(* CODESYS project SUZUKI.project
   Title: ifmCR711S_TemplateProject
   Company: ifm electronic
   Version: 2.4.13.0
   Description: Project template with CR711S configured 2.25MByte Standard 2.25MByte Safety

Project tree, tasks and I/O mapping:
  StandardPLC : CR711S Standard, ifm electronic, order no. CR711S, version 3.0.0.1
    application Application
      libraries: Standard, * (System); Util, * (System); SysMem, * (System); ifmR360-3, 1.1.1.0 (ifm electronic); SysTimeCore, 3.5.5.0 (System); SysFile, 3.5.9.0 (System); SysCom, 3.5.5.0 (System); ifmOutHBridge, 2.3.0.0 (ifm electronic); CAA CiA 405, 3.5.8.0 (CAA Technical Workgroup); TCP, 3.5.9.50 (3S - Smart Software Solutions GmbH)
      task Tarea_Can (cyclic, interval t#10ms, priority 0) calls nothing
      task Tarea_Codigo (cyclic, interval t#20ms, priority 1, watchdog t#200ms x 1) calls PLC_PRG
      CÓDIGO/
        program SALIDAS [ST]
        Seguridades/
          program Laser_Seguridad [ST]
          program Setas_Seguridad [ST]
          program Campos_Laser [ST]
        program SUPERVISOR [ST]
        Data types/
          data type AccionLevas
          data type ENTRADAS_PLC
          data type EstadoSecuenciaCarga
          data type CamposLaser
          data type ControlVelocidad
          data type ENTRADAS_AGV
          data type SALIDAS_PLC
          data type OperativaARealizar
          data type EstadoEframe
          data type VelocidadPorTramo
        AUX_IFM/
          function block fb_InputAddConf_sp_ST_V02 [FBD]
          function block fb_OutputGroupAddConf_sp_ST_V02 [FBD]
          function block fb_OutputAnaAddConf_sp_ST_V02 [FBD]
          function block fb_OutputAddConf_sp_ST_V02 [FBD]
        program ESTADOS [ST]
        Sub ACCIONES/
          program ACC03_ControlLevas [ST]
          program ACC00_SalidasDesactivadas [ST]
          program ACC02_ControlAutomatico [ST]
          program ACC01_ControlManual [ST]
        program IMAGENES [ST]
        program PLC_PRG [ST]
        program PARAMETRIZACION [ST]
        Sub Comunicacion/
          program C41 [ST]
          function block COM00_DispositivoCAN_FB [ST]
          program C40 [ST]
        Sub Temporizacion/
          program TEMP00_TiempoInicio [ST]
        program ACCIONES [ST]
        program COMUNICACION_CAN [ST]
        IO/
          program OUT01_WIRED_OUTPUTS [ST]
          program IN01_WIRED_INPUTS [ST]
        Sub Dispositivos/
          function block DISP01_CntrlExtensionGeneral_FB [ST]
          program DISP02_Indicadores [ST]
          program DISP03_EncoderTeaching [ST]
      Global Variables/
        global variables Variables_globales_persistentes
        data type MatrizPDO
        data type MatrizPDOUSINT
        data type SpCanOpenNode
        global variables Global_Variables
      Visualizaciones/
        trace Anomalia (task Tarea_Codigo): COMUNICACION_CAN.O_EstadoCAN.0
    Communication : Communication, ifm electronic, version 3.0.0.1
      Ethernet : Ethernet, ifm electronic, version 3.0.0.1
      CAN : CAN, ifm electronic, version 3.0.0.1
        ifmCANbus : ifmCANbus, ifm electronic, version 1.0.0.0
            settings: NetID = 2
          CANopen_Manager : CANopen_Manager, 3S - Smart Software Solutions GmbH, version 3.5.16.0
              settings: Sync CycleTime in Microseconds = 10000; Enable Sync generation = TRUE; Synchronous Window Length = 201010; NMT Start All = TRUE; Heartbeat in Milliseconds = 100; Heartbeat Node ID = 1; CANopen NodeID = 1; ConfigVersion = 50659584
            UCD_Encoder_Series : UCD Encoder Series, Posital GmbH, order no. UCD-CA01B-xxxx-xxxx-xxx, version Revision=16#00010000, FileVersion=1.1, File=UCD-CAx1B-xxxx-xxxx-xxx_V1R4.eds
                settings: General Options.Optional Device = TRUE; General Options.Reset Node = FALSE; NODEIDSAVED = 32; SDO Timeout = 1000000; PDO_Autoconfig = FALSE; EXPERTSETTINGS = True; Sync-General Parameters.Sync-COBID = 16#00000080; Sync-General Parameters.Communication Cycle Period = 16#00002710 usec; Synchronous Window Length = 16#00031132; SubIndex for reset node = 1; Emergency-General Parameters.Emergency enabled = FALSE; Emergency-General Parameters.Emergency COBID = 16#000000A0; Heartbeat-Producer Time = 100; PDO 16#1800.COBID = 16#000001A0; Process by CANopenManager = TRUE; PDO 16#1801.COBID = 16#000002A0; PDO 16#1801.Transmission Type = 16#01; Process by CANopenManager = TRUE; Heartbeat-Consuming1.Heartbeat-Time = 150 ms; Position value.Subindex = 16#00; Position value.Subindex = 16#00; SDO List.Set COB-ID sync.Index = 16#1005; SDO List.Set COB-ID sync.Subindex = 16#00; SDO List.Set COB-ID sync.Value = 16#00000080; SDO List.Set COB-ID sync.Size = 32; SDO List.Set COB-ID sync.AbortIfError = FALSE; SDO List.Set COB-ID sync.JumpToLine = FALSE; SDO List.Set COB-ID sync.Line = 0; SDO List.Set communication cycle period.Index = 16#1006; SDO List.Set communication cycle period.Subindex = 16#00; SDO List.Set communication cycle period.Value = 16#00002710; SDO List.Set communication cycle period.Size = 32; SDO List.Set communication cycle period.AbortIfError = FALSE; SDO List.Set communication cycle period.JumpToLine = FALSE; SDO List.Set communication cycle period.Line = 0; SDO List.Set synchronous window length.Index = 16#1007; SDO List.Set synchronous window length.Subindex = 16#00; SDO List.Set synchronous window length.Value = 16#00031132; SDO List.Set synchronous window length.Size = 32; SDO List.Set synchronous window length.AbortIfError = FALSE;
                  SDO List.Set synchronous window length.JumpToLine = FALSE; SDO List.Set synchronous window length.Line = 0; SDO List.Disable TIME.Index = 16#1012; SDO List.Disable TIME.Subindex = 16#00; SDO List.Disable TIME.Value = 16#00000100; SDO List.Disable TIME.Size = 32; SDO List.Disable TIME.AbortIfError = FALSE; SDO List.Disable TIME.JumpToLine = FALSE; SDO List.Disable TIME.Line = 0; SDO List.Set Guardtime.Index = 16#100C; SDO List.Set Guardtime.Subindex = 16#00; SDO List.Set Guardtime.Value = 16#00000000; SDO List.Set Guardtime.Size = 16; SDO List.Set Guardtime.AbortIfError = FALSE; SDO List.Set Guardtime.JumpToLine = FALSE; SDO List.Set Guardtime.Line = 0; SDO List.Set Lifetime.Index = 16#100D; SDO List.Set Lifetime.Subindex = 16#00; SDO List.Set Lifetime.Value = 16#00000000; SDO List.Set Lifetime.Size = 8; SDO List.Set Lifetime.AbortIfError = FALSE; SDO List.Set Lifetime.JumpToLine = FALSE; SDO List.Set Lifetime.Line = 0; SDO List.Set Heartbeat Consumer.Index = 16#1016; SDO List.Set Heartbeat Consumer.Subindex = 16#01; SDO List.Set Heartbeat Consumer.Value = 16#00010096; SDO List.Set Heartbeat Consumer.Size = 32; SDO List.Set Heartbeat Consumer.AbortIfError = FALSE; SDO List.Set Heartbeat Consumer.JumpToLine = FALSE; SDO List.Set Heartbeat Consumer.Line = 0; SDO List.Set Heartbeat Producer.Index = 16#1017; SDO List.Set Heartbeat Producer.Subindex = 16#00; SDO List.Set Heartbeat Producer.Value = 16#00000064; SDO List.Set Heartbeat Producer.Size = 16; SDO List.Set Heartbeat Producer.AbortIfError = FALSE; SDO List.Set Heartbeat Producer.JumpToLine = FALSE; SDO List.Set Heartbeat Producer.Line = 0; SDO List.Disable PDO.Index = 16#1800; SDO List.Disable PDO.Subindex = 16#01; SDO List.Disable PDO.Value = 16#800001A0;
                  SDO List.Disable PDO.Size = 32; SDO List.Disable PDO.AbortIfError = FALSE; SDO List.Disable PDO.JumpToLine = FALSE; SDO List.Disable PDO.Line = 0; SDO List.Set transmission type.Index = 16#1800; SDO List.Set transmission type.Subindex = 16#02; SDO List.Set transmission type.Value = 16#FE; SDO List.Set transmission type.Size = 8; SDO List.Set transmission type.AbortIfError = FALSE; SDO List.Set transmission type.JumpToLine = FALSE; SDO List.Set transmission type.Line = 0; SDO List.Set inhibit time.Index = 16#1800; SDO List.Set inhibit time.Subindex = 16#03; SDO List.Set inhibit time.Value = 16#0000; SDO List.Set inhibit time.Size = 16; SDO List.Set inhibit time.AbortIfError = FALSE; SDO List.Set inhibit time.JumpToLine = FALSE; SDO List.Set inhibit time.Line = 0; SDO List.Set event time.Index = 16#1800; SDO List.Set event time.Subindex = 16#05; SDO List.Set event time.Value = 16#0000; SDO List.Set event time.Size = 16; SDO List.Set event time.AbortIfError = FALSE; SDO List.Set event time.JumpToLine = FALSE; SDO List.Set event time.Line = 0; SDO List.Clear pdo mapping.Index = 16#1A00; SDO List.Clear pdo mapping.Subindex = 16#00; SDO List.Clear pdo mapping.Value = 16#0; SDO List.Clear pdo mapping.Size = 8; SDO List.Clear pdo mapping.AbortIfError = FALSE; SDO List.Clear pdo mapping.JumpToLine = FALSE; SDO List.Clear pdo mapping.Line = 0; SDO List.Set Mapping.Index = 16#1A00; SDO List.Set Mapping.Subindex = 16#01; SDO List.Set Mapping.Value = 16#60040020; SDO List.Set Mapping.Size = 32; SDO List.Set Mapping.AbortIfError = FALSE; SDO List.Set Mapping.JumpToLine = FALSE; SDO List.Set Mapping.Line = 0; SDO List.Set number of mappings.Index = 16#1A00;
                  SDO List.Set number of mappings.Subindex = 16#00; SDO List.Set number of mappings.Value = 16#01; SDO List.Set number of mappings.Size = 8; SDO List.Set number of mappings.AbortIfError = FALSE; SDO List.Set number of mappings.JumpToLine = FALSE; SDO List.Set number of mappings.Line = 0; SDO List.Set and enable COB-ID.Index = 16#1800; SDO List.Set and enable COB-ID.Subindex = 16#01; SDO List.Set and enable COB-ID.Value = 16#000001A0; SDO List.Set and enable COB-ID.Size = 32; SDO List.Set and enable COB-ID.AbortIfError = FALSE; SDO List.Set and enable COB-ID.JumpToLine = FALSE; SDO List.Set and enable COB-ID.Line = 0; SDO List.Disable PDO.Index = 16#1801; SDO List.Disable PDO.Subindex = 16#01; SDO List.Disable PDO.Value = 16#800002A0; SDO List.Disable PDO.Size = 32; SDO List.Disable PDO.AbortIfError = FALSE; SDO List.Disable PDO.JumpToLine = FALSE; SDO List.Disable PDO.Line = 0; SDO List.Set transmission type.Index = 16#1801; SDO List.Set transmission type.Subindex = 16#02; SDO List.Set transmission type.Value = 16#01; SDO List.Set transmission type.Size = 8; SDO List.Set transmission type.AbortIfError = FALSE; SDO List.Set transmission type.JumpToLine = FALSE; SDO List.Set transmission type.Line = 0; SDO List.Set inhibit time.Index = 16#1801; SDO List.Set inhibit time.Subindex = 16#03; SDO List.Set inhibit time.Value = 16#0000; SDO List.Set inhibit time.Size = 16; SDO List.Set inhibit time.AbortIfError = FALSE; SDO List.Set inhibit time.JumpToLine = FALSE; SDO List.Set inhibit time.Line = 0; SDO List.Set event time.Index = 16#1801; SDO List.Set event time.Subindex = 16#05; SDO List.Set event time.Value = 16#0000; SDO List.Set event time.Size = 16; SDO List.Set event time.AbortIfError = FALSE; SDO List.Set event time.JumpToLine = FALSE;
                  SDO List.Set event time.Line = 0; SDO List.Clear pdo mapping.Index = 16#1A01; SDO List.Clear pdo mapping.Subindex = 16#00; SDO List.Clear pdo mapping.Value = 16#0; SDO List.Clear pdo mapping.Size = 8; SDO List.Clear pdo mapping.AbortIfError = FALSE; SDO List.Clear pdo mapping.JumpToLine = FALSE; SDO List.Clear pdo mapping.Line = 0; SDO List.Set Mapping.Index = 16#1A01; SDO List.Set Mapping.Subindex = 16#01; SDO List.Set Mapping.Value = 16#60040020; SDO List.Set Mapping.Size = 32; SDO List.Set Mapping.AbortIfError = FALSE; SDO List.Set Mapping.JumpToLine = FALSE; SDO List.Set Mapping.Line = 0; SDO List.Set number of mappings.Index = 16#1A01; SDO List.Set number of mappings.Subindex = 16#00; SDO List.Set number of mappings.Value = 16#01; SDO List.Set number of mappings.Size = 8; SDO List.Set number of mappings.AbortIfError = FALSE; SDO List.Set number of mappings.JumpToLine = FALSE; SDO List.Set number of mappings.Line = 0; SDO List.Set and enable COB-ID.Index = 16#1801; SDO List.Set and enable COB-ID.Subindex = 16#01; SDO List.Set and enable COB-ID.Value = 16#000002A0; SDO List.Set and enable COB-ID.Size = 32; SDO List.Set and enable COB-ID.AbortIfError = FALSE; SDO List.Set and enable COB-ID.JumpToLine = FALSE; SDO List.Set and enable COB-ID.Line = 0; ConfigVersion = 50659584
                unmapped channels: Position value, Position value
    HMI : HMI, ifm electronic, version 3.0.0.1
      User_LEDs : User_LEDs, ifm electronic, version 3.0.0.1
          input  UserLED0_I : LED_IEC_B_INPUT_MAPPING_TYPE  // UserLED0_I
          input  UserLED1_I : LED_IEC_B_INPUT_MAPPING_TYPE  // UserLED1_I
          input  UserLED2_I : LED_IEC_B_INPUT_MAPPING_TYPE  // UserLED2_I
          input  UserLED3_I : LED_IEC_B_INPUT_MAPPING_TYPE  // UserLED3_I
          output UserLED0_Q : LED_IEC_B_OUTPUT_MAPPING_TYPE  // User LED 0
          output UserLED1_Q : LED_IEC_B_OUTPUT_MAPPING_TYPE  // User LED 1
          output UserLED2_Q : LED_IEC_B_OUTPUT_MAPPING_TYPE  // User LED 2
          output UserLED3_Q : LED_IEC_B_OUTPUT_MAPPING_TYPE  // User LED 3
    Local_IO : Local_IO, ifm electronic, version 3.0.0.1
      Outputs : Outputs, ifm electronic, version 3.0.0.1
          input  OUT0006_I : OUT_PWM_40_BRIDGE_A_INPUT_MAPPING_TYPE  // OUT0006_I
          input  OUT0106_I : OUT_PWM_40_BRIDGE_A_INPUT_MAPPING_TYPE  // OUT0106_I
          input  OUT0206_I : OUT_PWM_40_BRIDGE_A_INPUT_MAPPING_TYPE  // OUT0206_I
          input  OUT0008_I : OUT_PWM_40_A_INPUT_MAPPING_TYPE  // OUT0008_I
          input  OUT0108_I : OUT_PWM_40_A_INPUT_MAPPING_TYPE  // OUT0108_I
          input  OUT0208_I : OUT_PWM_40_A_INPUT_MAPPING_TYPE  // OUT0208_I
          input  OUT0000_I : OUT_PWM_25_A_INPUT_MAPPING_TYPE  // OUT0000_I
          input  OUT0002_I : OUT_PWM_25_A_INPUT_MAPPING_TYPE  // OUT0002_I
          input  OUT0004_I : OUT_PWM_25_A_INPUT_MAPPING_TYPE  // OUT0004_I
          input  OUT0100_I : OUT_PWM_25_A_INPUT_MAPPING_TYPE  // OUT0100_I
          input  OUT0102_I : OUT_PWM_25_A_INPUT_MAPPING_TYPE  // OUT0102_I
          input  OUT0104_I : OUT_PWM_25_A_INPUT_MAPPING_TYPE  // OUT0104_I
          input  OUT0200_I : OUT_PWM_25_A_INPUT_MAPPING_TYPE  // OUT0200_I
          input  OUT0202_I : OUT_PWM_25_A_INPUT_MAPPING_TYPE  // OUT0202_I
          input  OUT0204_I : OUT_PWM_25_A_INPUT_MAPPING_TYPE  // OUT0204_I
          input  OUT3001_I : OUT_VOLTAGE_A_INPUT_MAPPING_TYPE  // OUT3001_I
          input  OUT3000_I : OUT_SUPPLY_A_INPUT_MAPPING_TYPE  // OUT3000_I
          input  OUT0001_I : OUT_PWM_25_B_INPUT_MAPPING_TYPE  // OUT0001_I
          input  OUT0003_I : OUT_PWM_25_B_INPUT_MAPPING_TYPE  // OUT0003_I
          input  OUT0005_I : OUT_PWM_25_B_INPUT_MAPPING_TYPE  // OUT0005_I
          input  OUT0101_I : OUT_PWM_25_B_INPUT_MAPPING_TYPE  // OUT0101_I
          input  OUT0103_I : OUT_PWM_25_B_INPUT_MAPPING_TYPE  // OUT0103_I
          input  OUT0105_I : OUT_PWM_25_B_INPUT_MAPPING_TYPE  // OUT0105_I
          input  OUT0201_I : OUT_PWM_25_B_INPUT_MAPPING_TYPE  // OUT0201_I
          input  OUT0203_I : OUT_PWM_25_B_INPUT_MAPPING_TYPE  // OUT0203_I
          input  OUT0205_I : OUT_PWM_25_B_INPUT_MAPPING_TYPE  // OUT0205_I
          input  OUT0007_I : OUT_PWM_40_BRIDGE_A_INPUT_MAPPING_TYPE  // OUT0007_I
          input  OUT0107_I : OUT_PWM_40_BRIDGE_A_INPUT_MAPPING_TYPE  // OUT0107_I
          input  OUT0207_I : OUT_PWM_40_BRIDGE_A_INPUT_MAPPING_TYPE  // OUT0207_I
          output OUT0006_Q : OUT_PWM_40_BRIDGE_A_OUTPUT_MAPPING_TYPE  // OUT0006_Q
          output OUT0106_Q : OUT_PWM_40_BRIDGE_A_OUTPUT_MAPPING_TYPE  // OUT0106_Q
          output OUT0206_Q : OUT_PWM_40_BRIDGE_A_OUTPUT_MAPPING_TYPE  // OUT0206_Q
          output OUT0008_Q : OUT_PWM_40_A_OUTPUT_MAPPING_TYPE  // OUT0008_Q
          output OUT0108_Q : OUT_PWM_40_A_OUTPUT_MAPPING_TYPE  // OUT0108_Q
          output OUT0208_Q : OUT_PWM_40_A_OUTPUT_MAPPING_TYPE  // OUT0208_Q
          output OUT0000_Q : OUT_PWM_25_A_OUTPUT_MAPPING_TYPE  // OUT0000_Q
          output OUT0002_Q : OUT_PWM_25_A_OUTPUT_MAPPING_TYPE  // OUT0002_Q
          output OUT0004_Q : OUT_PWM_25_A_OUTPUT_MAPPING_TYPE  // OUT0004_Q
          output OUT0100_Q : OUT_PWM_25_A_OUTPUT_MAPPING_TYPE  // OUT0100_Q
          output OUT0102_Q : OUT_PWM_25_A_OUTPUT_MAPPING_TYPE  // OUT0102_Q
          output OUT0104_Q : OUT_PWM_25_A_OUTPUT_MAPPING_TYPE  // OUT0104_Q
          output OUT0200_Q : OUT_PWM_25_A_OUTPUT_MAPPING_TYPE  // OUT0200_Q
          output OUT0202_Q : OUT_PWM_25_A_OUTPUT_MAPPING_TYPE  // OUT0202_Q
          output OUT0204_Q : OUT_PWM_25_A_OUTPUT_MAPPING_TYPE  // OUT0204_Q
          output OUT3001_Q : OUT_VOLTAGE_A_OUTPUT_MAPPING_TYPE  // OUT3001_Q
          output OUT3000_Q : OUT_SUPPLY_A_OUTPUT_MAPPING_TYPE  // OUT3000_Q
          output OUT0001_Q : OUT_PWM_25_B_OUTPUT_MAPPING_TYPE  // OUT0001_Q
          output OUT0003_Q : OUT_PWM_25_B_OUTPUT_MAPPING_TYPE  // OUT0003_Q
          output OUT0005_Q : OUT_PWM_25_B_OUTPUT_MAPPING_TYPE  // OUT0005_Q
          output OUT0101_Q : OUT_PWM_25_B_OUTPUT_MAPPING_TYPE  // OUT0101_Q
          output OUT0103_Q : OUT_PWM_25_B_OUTPUT_MAPPING_TYPE  // OUT0103_Q
          output OUT0105_Q : OUT_PWM_25_B_OUTPUT_MAPPING_TYPE  // OUT0105_Q
          output OUT0201_Q : OUT_PWM_25_B_OUTPUT_MAPPING_TYPE  // OUT0201_Q
          output OUT0203_Q : OUT_PWM_25_B_OUTPUT_MAPPING_TYPE  // OUT0203_Q
          output OUT0205_Q : OUT_PWM_25_B_OUTPUT_MAPPING_TYPE  // OUT0205_Q
          output OUT0007_Q : OUT_PWM_40_BRIDGE_A_OUTPUT_MAPPING_TYPE  // OUT0007_Q
          output OUT0107_Q : OUT_PWM_40_BRIDGE_A_OUTPUT_MAPPING_TYPE  // OUT0107_Q
          output OUT0207_Q : OUT_PWM_40_BRIDGE_A_OUTPUT_MAPPING_TYPE  // OUT0207_Q
      System_Inputs : System_Inputs, ifm electronic, version 3.0.0.1
          input  VBB30 : IN_SYSTEM_VOLTAGE_INPUT_MAPPING_TYPE  // VBB30
          input  VBB15 : IN_SYSTEM_VOLTAGE_INPUT_MAPPING_TYPE  // VBB15
          input  TemperatureBoard0 : IN_TEMPERATURE_INPUT_MAPPING_TYPE  // TemperatureBoard0
          input  TemperatureChip0 : IN_TEMPERATURE_INPUT_MAPPING_TYPE  // TemperatureChip0
      Inputs : Inputs, ifm electronic, version 3.0.0.1
          input  IN0100_I : IN_MULTIFUNCTION_A_INPUT_MAPPING_TYPE  // IN0100_I
          input  IN0101_I : IN_MULTIFUNCTION_A_INPUT_MAPPING_TYPE  // IN0101_I
          input  IN0102_I : IN_MULTIFUNCTION_A_INPUT_MAPPING_TYPE  // IN0102_I
          input  IN0103_I : IN_MULTIFUNCTION_A_INPUT_MAPPING_TYPE  // IN0103_I
          input  IN0200_I : IN_MULTIFUNCTION_A_INPUT_MAPPING_TYPE  // IN0200_I
          input  IN0201_I : IN_MULTIFUNCTION_A_INPUT_MAPPING_TYPE  // IN0201_I
          input  IN0202_I : IN_MULTIFUNCTION_A_INPUT_MAPPING_TYPE  // IN0202_I
          input  IN0203_I : IN_MULTIFUNCTION_A_INPUT_MAPPING_TYPE  // IN0203_I
          input  IN0600_I : IN_MULTIFUNCTION_A_INPUT_MAPPING_TYPE  // IN0600_I
          input  IN0601_I : IN_MULTIFUNCTION_A_INPUT_MAPPING_TYPE  // IN0601_I
          input  IN0602_I : IN_MULTIFUNCTION_A_INPUT_MAPPING_TYPE  // IN0602_I
          input  IN0603_I : IN_MULTIFUNCTION_A_INPUT_MAPPING_TYPE  // IN0603_I
          input  IN0700_I : IN_MULTIFUNCTION_A_INPUT_MAPPING_TYPE  // IN0700_I
          input  IN0701_I : IN_MULTIFUNCTION_A_INPUT_MAPPING_TYPE  // IN0701_I
          input  IN0702_I : IN_MULTIFUNCTION_A_INPUT_MAPPING_TYPE  // IN0702_I
          input  IN0703_I : IN_MULTIFUNCTION_A_INPUT_MAPPING_TYPE  // IN0703_I
          input  IN0400_I : IN_RESISTOR_A_INPUT_MAPPING_TYPE  // IN0400_I
          input  IN0401_I : IN_RESISTOR_A_INPUT_MAPPING_TYPE  // IN0401_I
          input  IN0900_I : IN_RESISTOR_A_INPUT_MAPPING_TYPE  // IN0900_I
          input  IN0901_I : IN_RESISTOR_A_INPUT_MAPPING_TYPE  // IN0901_I
          input  IN0300_I : IN_DIGITAL_B_INPUT_MAPPING_TYPE  // IN0300_I
          input  IN0301_I : IN_DIGITAL_B_INPUT_MAPPING_TYPE  // IN0301_I
          input  IN0800_I : IN_DIGITAL_B_INPUT_MAPPING_TYPE  // IN0800_I
          input  IN0801_I : IN_DIGITAL_B_INPUT_MAPPING_TYPE  // IN0801_I
          input  COM_RESET_I : IN_COMMUNICATION_RESET_INPUT_MAPPING_TYPE  // COM_RESET_I
          input  IN0000_I : IN_FREQUENCY_B_CHANNEL_A_INPUT_MAPPING_TYPE  // IN0000_I
          input  IN0002_I : IN_FREQUENCY_B_CHANNEL_A_INPUT_MAPPING_TYPE  // IN0002_I
          input  IN0500_I : IN_FREQUENCY_B_CHANNEL_A_INPUT_MAPPING_TYPE  // IN0500_I
          input  IN0502_I : IN_FREQUENCY_B_CHANNEL_A_INPUT_MAPPING_TYPE  // IN0502_I
          input  IN0001_I : IN_FREQUENCY_B_CHANNEL_B_INPUT_MAPPING_TYPE  // IN0001_I
          input  IN0003_I : IN_FREQUENCY_B_CHANNEL_B_INPUT_MAPPING_TYPE  // IN0003_I
          input  IN0501_I : IN_FREQUENCY_B_CHANNEL_B_INPUT_MAPPING_TYPE  // IN0501_I
          input  IN0503_I : IN_FREQUENCY_B_CHANNEL_B_INPUT_MAPPING_TYPE  // IN0503_I
      System_Outputs : System_Outputs, ifm electronic, version 3.0.0.1
          input  VBB0_SW_I : OUT_GROUP_SWITCH_INPUT_MAPPING_TYPE  // VBB0_SW_I
          input  VBB1_SW_I : OUT_GROUP_SWITCH_INPUT_MAPPING_TYPE  // VBB1_SW_I
          input  VBB2_SW_I : OUT_GROUP_SWITCH_INPUT_MAPPING_TYPE  // VBB2_SW_I
          output VBB0_SW_Q : OUT_GROUP_SWITCH_OUTPUT_MAPPING_TYPE  // VBB0_SW_Q
          output VBB1_SW_Q : OUT_GROUP_SWITCH_OUTPUT_MAPPING_TYPE  // VBB1_SW_Q
          output VBB2_SW_Q : OUT_GROUP_SWITCH_OUTPUT_MAPPING_TYPE  // VBB2_SW_Q
          output SUPPLY_SWITCH_Q : OUT_SYS_SWITCH_OUTPUT_MAPPING_TYPE  // SUPPLY_SWITCH_Q
  SafetyPLC : CR711S SIL2, ifm electronic, order no. CR711S, version 3.0.0.1
    application Application
    Communication : Communication, ifm electronic, version 3.0.0.1
      Ethernet : Ethernet, ifm electronic, version 3.0.0.1
      CAN : CAN, ifm electronic, version 3.0.0.1
    HMI : HMI, ifm electronic, version 3.0.0.1
      User_LEDs : User_LEDs, ifm electronic, version 3.0.0.1
          input  UserLED0_I : LED_IEC_B_INPUT_MAPPING_TYPE  // UserLED0_I
          input  UserLED1_I : LED_IEC_B_INPUT_MAPPING_TYPE  // UserLED1_I
          input  UserLED2_I : LED_IEC_B_INPUT_MAPPING_TYPE  // UserLED2_I
          input  UserLED3_I : LED_IEC_B_INPUT_MAPPING_TYPE  // UserLED3_I
          output UserLED0_Q : LED_IEC_B_OUTPUT_MAPPING_TYPE  // User LED 0
          output UserLED1_Q : LED_IEC_B_OUTPUT_MAPPING_TYPE  // User LED 1
          output UserLED2_Q : LED_IEC_B_OUTPUT_MAPPING_TYPE  // User LED 2
          output UserLED3_Q : LED_IEC_B_OUTPUT_MAPPING_TYPE  // User LED 3
    Local_IO : Local_IO, ifm electronic, version 3.0.0.1
      System_Outputs : System_Outputs, ifm electronic, version 3.0.0.1
          input  VBB0_SW_I : OUT_GROUP_SWITCH_INPUT_MAPPING_TYPE  // VBB0_SW_I
          input  VBB1_SW_I : OUT_GROUP_SWITCH_INPUT_MAPPING_TYPE  // VBB1_SW_I
          input  VBB2_SW_I : OUT_GROUP_SWITCH_INPUT_MAPPING_TYPE  // VBB2_SW_I
          output VBB0_SW_Q : OUT_GROUP_SWITCH_OUTPUT_MAPPING_TYPE  // VBB0_SW_Q
          output VBB1_SW_Q : OUT_GROUP_SWITCH_OUTPUT_MAPPING_TYPE  // VBB1_SW_Q
          output VBB2_SW_Q : OUT_GROUP_SWITCH_OUTPUT_MAPPING_TYPE  // VBB2_SW_Q
          output SUPPLY_SWITCH_Q : OUT_SYS_SWITCH_OUTPUT_MAPPING_TYPE  // SUPPLY_SWITCH_Q
      Inputs : Inputs, ifm electronic, version 3.0.0.1
          input  IN0100_I : IN_MULTIFUNCTION_A_INPUT_MAPPING_TYPE  // IN0100_I
          input  IN0101_I : IN_MULTIFUNCTION_A_INPUT_MAPPING_TYPE  // IN0101_I
          input  IN0102_I : IN_MULTIFUNCTION_A_INPUT_MAPPING_TYPE  // IN0102_I
          input  IN0103_I : IN_MULTIFUNCTION_A_INPUT_MAPPING_TYPE  // IN0103_I
          input  IN0200_I : IN_MULTIFUNCTION_A_INPUT_MAPPING_TYPE  // IN0200_I
          input  IN0201_I : IN_MULTIFUNCTION_A_INPUT_MAPPING_TYPE  // IN0201_I
          input  IN0202_I : IN_MULTIFUNCTION_A_INPUT_MAPPING_TYPE  // IN0202_I
          input  IN0203_I : IN_MULTIFUNCTION_A_INPUT_MAPPING_TYPE  // IN0203_I
          input  IN0600_I : IN_MULTIFUNCTION_A_INPUT_MAPPING_TYPE  // IN0600_I
          input  IN0601_I : IN_MULTIFUNCTION_A_INPUT_MAPPING_TYPE  // IN0601_I
          input  IN0602_I : IN_MULTIFUNCTION_A_INPUT_MAPPING_TYPE  // IN0602_I
          input  IN0603_I : IN_MULTIFUNCTION_A_INPUT_MAPPING_TYPE  // IN0603_I
          input  IN0700_I : IN_MULTIFUNCTION_A_INPUT_MAPPING_TYPE  // IN0700_I
          input  IN0701_I : IN_MULTIFUNCTION_A_INPUT_MAPPING_TYPE  // IN0701_I
          input  IN0702_I : IN_MULTIFUNCTION_A_INPUT_MAPPING_TYPE  // IN0702_I
          input  IN0703_I : IN_MULTIFUNCTION_A_INPUT_MAPPING_TYPE  // IN0703_I
          input  IN0400_I : IN_RESISTOR_A_INPUT_MAPPING_TYPE  // IN0400_I
          input  IN0401_I : IN_RESISTOR_A_INPUT_MAPPING_TYPE  // IN0401_I
          input  IN0900_I : IN_RESISTOR_A_INPUT_MAPPING_TYPE  // IN0900_I
          input  IN0901_I : IN_RESISTOR_A_INPUT_MAPPING_TYPE  // IN0901_I
          input  IN0300_I : IN_DIGITAL_B_INPUT_MAPPING_TYPE  // IN0300_I
          input  IN0301_I : IN_DIGITAL_B_INPUT_MAPPING_TYPE  // IN0301_I
          input  IN0800_I : IN_DIGITAL_B_INPUT_MAPPING_TYPE  // IN0800_I
          input  IN0801_I : IN_DIGITAL_B_INPUT_MAPPING_TYPE  // IN0801_I
          input  COM_RESET_I : IN_COMMUNICATION_RESET_INPUT_MAPPING_TYPE  // COM_RESET_I
          input  IN0000_I : IN_FREQUENCY_B_CHANNEL_A_INPUT_MAPPING_TYPE  // IN0000_I
          input  IN0002_I : IN_FREQUENCY_B_CHANNEL_A_INPUT_MAPPING_TYPE  // IN0002_I
          input  IN0500_I : IN_FREQUENCY_B_CHANNEL_A_INPUT_MAPPING_TYPE  // IN0500_I
          input  IN0502_I : IN_FREQUENCY_B_CHANNEL_A_INPUT_MAPPING_TYPE  // IN0502_I
          input  IN0001_I : IN_FREQUENCY_B_CHANNEL_B_INPUT_MAPPING_TYPE  // IN0001_I
          input  IN0003_I : IN_FREQUENCY_B_CHANNEL_B_INPUT_MAPPING_TYPE  // IN0003_I
          input  IN0501_I : IN_FREQUENCY_B_CHANNEL_B_INPUT_MAPPING_TYPE  // IN0501_I
          input  IN0503_I : IN_FREQUENCY_B_CHANNEL_B_INPUT_MAPPING_TYPE  // IN0503_I
      System_Inputs : System_Inputs, ifm electronic, version 3.0.0.1
          input  VBB30 : IN_SYSTEM_VOLTAGE_INPUT_MAPPING_TYPE  // VBB30
          input  VBB15 : IN_SYSTEM_VOLTAGE_INPUT_MAPPING_TYPE  // VBB15
          input  TemperatureBoard0 : IN_TEMPERATURE_INPUT_MAPPING_TYPE  // TemperatureBoard0
          input  TemperatureChip0 : IN_TEMPERATURE_INPUT_MAPPING_TYPE  // TemperatureChip0
      Outputs : Outputs, ifm electronic, version 3.0.0.1
          input  OUT0006_I : OUT_PWM_40_BRIDGE_A_INPUT_MAPPING_TYPE  // OUT0006_I
          input  OUT0106_I : OUT_PWM_40_BRIDGE_A_INPUT_MAPPING_TYPE  // OUT0106_I
          input  OUT0206_I : OUT_PWM_40_BRIDGE_A_INPUT_MAPPING_TYPE  // OUT0206_I
          input  OUT0008_I : OUT_PWM_40_A_INPUT_MAPPING_TYPE  // OUT0008_I
          input  OUT0108_I : OUT_PWM_40_A_INPUT_MAPPING_TYPE  // OUT0108_I
          input  OUT0208_I : OUT_PWM_40_A_INPUT_MAPPING_TYPE  // OUT0208_I
          input  OUT0000_I : OUT_PWM_25_A_INPUT_MAPPING_TYPE  // OUT0000_I
          input  OUT0002_I : OUT_PWM_25_A_INPUT_MAPPING_TYPE  // OUT0002_I
          input  OUT0004_I : OUT_PWM_25_A_INPUT_MAPPING_TYPE  // OUT0004_I
          input  OUT0100_I : OUT_PWM_25_A_INPUT_MAPPING_TYPE  // OUT0100_I
          input  OUT0102_I : OUT_PWM_25_A_INPUT_MAPPING_TYPE  // OUT0102_I
          input  OUT0104_I : OUT_PWM_25_A_INPUT_MAPPING_TYPE  // OUT0104_I
          input  OUT0200_I : OUT_PWM_25_A_INPUT_MAPPING_TYPE  // OUT0200_I
          input  OUT0202_I : OUT_PWM_25_A_INPUT_MAPPING_TYPE  // OUT0202_I
          input  OUT0204_I : OUT_PWM_25_A_INPUT_MAPPING_TYPE  // OUT0204_I
          input  OUT3001_I : OUT_VOLTAGE_A_INPUT_MAPPING_TYPE  // OUT3001_I
          input  OUT3000_I : OUT_SUPPLY_A_INPUT_MAPPING_TYPE  // OUT3000_I
          input  OUT0001_I : OUT_PWM_25_B_INPUT_MAPPING_TYPE  // OUT0001_I
          input  OUT0003_I : OUT_PWM_25_B_INPUT_MAPPING_TYPE  // OUT0003_I
          input  OUT0005_I : OUT_PWM_25_B_INPUT_MAPPING_TYPE  // OUT0005_I
          input  OUT0101_I : OUT_PWM_25_B_INPUT_MAPPING_TYPE  // OUT0101_I
          input  OUT0103_I : OUT_PWM_25_B_INPUT_MAPPING_TYPE  // OUT0103_I
          input  OUT0105_I : OUT_PWM_25_B_INPUT_MAPPING_TYPE  // OUT0105_I
          input  OUT0201_I : OUT_PWM_25_B_INPUT_MAPPING_TYPE  // OUT0201_I
          input  OUT0203_I : OUT_PWM_25_B_INPUT_MAPPING_TYPE  // OUT0203_I
          input  OUT0205_I : OUT_PWM_25_B_INPUT_MAPPING_TYPE  // OUT0205_I
          input  OUT0007_I : OUT_PWM_40_BRIDGE_A_INPUT_MAPPING_TYPE  // OUT0007_I
          input  OUT0107_I : OUT_PWM_40_BRIDGE_A_INPUT_MAPPING_TYPE  // OUT0107_I
          input  OUT0207_I : OUT_PWM_40_BRIDGE_A_INPUT_MAPPING_TYPE  // OUT0207_I
          output OUT0006_Q : OUT_PWM_40_BRIDGE_A_OUTPUT_MAPPING_TYPE  // OUT0006_Q
          output OUT0106_Q : OUT_PWM_40_BRIDGE_A_OUTPUT_MAPPING_TYPE  // OUT0106_Q
          output OUT0206_Q : OUT_PWM_40_BRIDGE_A_OUTPUT_MAPPING_TYPE  // OUT0206_Q
          output OUT0008_Q : OUT_PWM_40_A_OUTPUT_MAPPING_TYPE  // OUT0008_Q
          output OUT0108_Q : OUT_PWM_40_A_OUTPUT_MAPPING_TYPE  // OUT0108_Q
          output OUT0208_Q : OUT_PWM_40_A_OUTPUT_MAPPING_TYPE  // OUT0208_Q
          output OUT0000_Q : OUT_PWM_25_A_OUTPUT_MAPPING_TYPE  // OUT0000_Q
          output OUT0002_Q : OUT_PWM_25_A_OUTPUT_MAPPING_TYPE  // OUT0002_Q
          output OUT0004_Q : OUT_PWM_25_A_OUTPUT_MAPPING_TYPE  // OUT0004_Q
          output OUT0100_Q : OUT_PWM_25_A_OUTPUT_MAPPING_TYPE  // OUT0100_Q
          output OUT0102_Q : OUT_PWM_25_A_OUTPUT_MAPPING_TYPE  // OUT0102_Q
          output OUT0104_Q : OUT_PWM_25_A_OUTPUT_MAPPING_TYPE  // OUT0104_Q
          output OUT0200_Q : OUT_PWM_25_A_OUTPUT_MAPPING_TYPE  // OUT0200_Q
          output OUT0202_Q : OUT_PWM_25_A_OUTPUT_MAPPING_TYPE  // OUT0202_Q
          output OUT0204_Q : OUT_PWM_25_A_OUTPUT_MAPPING_TYPE  // OUT0204_Q
          output OUT3001_Q : OUT_VOLTAGE_A_OUTPUT_MAPPING_TYPE  // OUT3001_Q
          output OUT3000_Q : OUT_SUPPLY_A_OUTPUT_MAPPING_TYPE  // OUT3000_Q
          output OUT0001_Q : OUT_PWM_25_B_OUTPUT_MAPPING_TYPE  // OUT0001_Q
          output OUT0003_Q : OUT_PWM_25_B_OUTPUT_MAPPING_TYPE  // OUT0003_Q
          output OUT0005_Q : OUT_PWM_25_B_OUTPUT_MAPPING_TYPE  // OUT0005_Q
          output OUT0101_Q : OUT_PWM_25_B_OUTPUT_MAPPING_TYPE  // OUT0101_Q
          output OUT0103_Q : OUT_PWM_25_B_OUTPUT_MAPPING_TYPE  // OUT0103_Q
          output OUT0105_Q : OUT_PWM_25_B_OUTPUT_MAPPING_TYPE  // OUT0105_Q
          output OUT0201_Q : OUT_PWM_25_B_OUTPUT_MAPPING_TYPE  // OUT0201_Q
          output OUT0203_Q : OUT_PWM_25_B_OUTPUT_MAPPING_TYPE  // OUT0203_Q
          output OUT0205_Q : OUT_PWM_25_B_OUTPUT_MAPPING_TYPE  // OUT0205_Q
          output OUT0007_Q : OUT_PWM_40_BRIDGE_A_OUTPUT_MAPPING_TYPE  // OUT0007_Q
          output OUT0107_Q : OUT_PWM_40_BRIDGE_A_OUTPUT_MAPPING_TYPE  // OUT0107_Q
          output OUT0207_Q : OUT_PWM_40_BRIDGE_A_OUTPUT_MAPPING_TYPE  // OUT0207_Q
  CR711S : CR711S, ifm electronic, order no. CR711S, version 3.0.0.1
  Project Information/
    function GetNumberProperty [ST]
    function GetVersionProperty [ST]
    function GetBooleanProperty [ST]
    function GetTextProperty [ST]
    function GetTextProperty2 [ST]
    function GetTitle [ST]
    function GetCompany [ST]
    function GetVersion [ST]
  text list GlobalTextList
*)

// StandardPLC/Application/CÓDIGO/Data types/AccionLevas
TYPE AccionLevas : (subir, bajar,apagado);
END_TYPE

// StandardPLC/Application/CÓDIGO/Data types/ENTRADAS_PLC
TYPE ENTRADAS_PLC :
STRUCT
	Manual_RecogerBrazo			:BOOL;
	Manual_ExtenderBrazo        :BOOL;
	
	InductivoSubirLevas         :BOOL;   
	InductivoBajarLevas         :BOOL;
	
	DeteccionCarga1             :BOOL;   //Inductivo deteccion de carga 1
	DeteccionCarga2             :BOOL;   //Inductivo deteccion de carga 2
	DeteccionCargaExt       	:BOOL;   //Inductivo deteccion de carga cuando esta a extender el brazo
	
	ParadaPrecisaBrazo          :BOOL;   //Fotocelula Brazo
	ParadaPrecisaEFrame         :BOOL;   //Fotocelula E-Frame
	
	InductivoBrazoRec           :BOOL;   //Inductivo husillo 4
	InductivoBrazoExt           :BOOL;   //Inductivo husillo 5
	
	SetaEmergenciaIN1			:BOOL;
	SetaEmergenciaIN2			:BOOL;
	
	BotonRearme					:BOOL;
	
	Laser_OSSD1					:BOOL;
	Laser_OSSD2					:BOOL;
	
	ModoAutomatico				:BOOL;
	
	Modo_Degradado				:BOOL;
	
	Manual_SubirLevas			:BOOL;
	Manual_BajarLevas			:BOOL;
END_STRUCT
END_TYPE

// StandardPLC/Application/Global Variables/MatrizPDO
TYPE MatrizPDO :
STRUCT
	Matriz		:ARRAY[0..7] OF BYTE;
END_STRUCT
END_TYPE

// StandardPLC/Application/CÓDIGO/Data types/EstadoSecuenciaCarga
TYPE EstadoSecuenciaCarga : (indeterminado, descargado, cargado);
END_TYPE

// StandardPLC/Application/CÓDIGO/Data types/CamposLaser
TYPE CamposLaser : (Bumper, Ext_con_carga_1600, Ext_con_carga_1800, Ext_sin_carga);
END_TYPE

// StandardPLC/Application/CÓDIGO/Data types/ControlVelocidad
TYPE ControlVelocidad : (A_Recoger, A_Extender, A_Parar,M_Recoger, M_Extender, M_Parar, Laser_Parar, Setas_Parar, Anomalia_Parar, Retener_Auto);
END_TYPE

// StandardPLC/Application/Global Variables/MatrizPDOUSINT
TYPE MatrizPDOUSINT :
STRUCT
	Matriz		:ARRAY[0..7] OF USINT;
END_STRUCT
END_TYPE

// StandardPLC/Application/CÓDIGO/Data types/ENTRADAS_AGV
TYPE ENTRADAS_AGV :
STRUCT
	Manual				:BOOL;
	Rearmar				:BOOL;
	EmergenciasAGV		:BOOL;
	Habilitar			:BOOL;
	OrdenCarga			:BOOL;
	OrdenDescarga		:BOOL;
	ForzarBumper        :BOOL;
	OrdenDescargaB		:BOOL;
END_STRUCT
END_TYPE

// StandardPLC/Application/CÓDIGO/Data types/SALIDAS_PLC
TYPE SALIDAS_PLC :
STRUCT
	Consigna				:INT;
	
	SubirLevas				:BOOL;
	BajarLevas				:BOOL;
	
	Contactor				:BOOL;
	Contactor2				:BOOL;
	
	Eletrofreno				:BOOL;
	
	ContactorHabVariador	:BOOL;
	
	LuzAmarillo 			:BOOL;
	LuzRojo					:BOOL;
	LuzVerde				:BOOL;
	Acustico				:BOOL;
	LuzBotonRearme			:BOOL;
	
	ExtrairBrazo			:BOOL;
	RetrairBrazo			:BOOL;
	
	SeguroLaser				:BOOL;
	SeguroSetas				:BOOL;
	Seta_CAN				:BOOL;
	
	LaserA					:BOOL;
	LaserB					:BOOL;
	LaserC					:BOOL;
	LaserAA					:BOOL;		//A'
	LaserBB					:BOOL;		//B'
	LaserCC					:BOOL;		//C'
	
	SetaEmergenciaOUT1		:SAFEBOOL;
	SetaEmergenciaOUT2		:SAFEBOOL;
	
	Ch1_ReleSeguridad		:BOOL;
	Ch2_ReleSeguridad		:BOOL;
END_STRUCT
END_TYPE

// StandardPLC/Application/CÓDIGO/Data types/OperativaARealizar
TYPE OperativaARealizar : (init_descargado, init_cargado, indeterminado_OPT, init_cargado_B);
END_TYPE

// StandardPLC/Application/CÓDIGO/Data types/EstadoEframe
TYPE EstadoEframe : (Identificar, Reposo, Automatico, Anomalia, Manual, Degradado, Reinicio);
END_TYPE

// StandardPLC/Application/Global Variables/SpCanOpenNode
TYPE SpCanOpenNode :
STRUCT
	nStatus		:INT;
	ucNodeNr	:BYTE;
END_STRUCT
END_TYPE

// StandardPLC/Application/CÓDIGO/Data types/VelocidadPorTramo
TYPE VelocidadPorTramo : (E_Cargado_Tramo1, E_Cargado_Tramo2, E_Cargado_Tramo3, E_Descargado_Tramo1, E_Descargado_Tramo2, E_Descargado_Tramo3, R_Cargado_Tramo1, R_Cargado_Tramo2, R_Cargado_Tramo3, R_Descargado_Tramo1, R_Descargado_Tramo2, SinConsigna);
END_TYPE

// StandardPLC/Application/Global Variables/Variables_globales_persistentes
VAR_GLOBAL PERSISTENT RETAIN	
	gEncoder_Absoluto				:UDINT; 
	gEncoder_AbsolutoExtendido		:UDINT; 
	gEncoder_OperativaB				:UDINT; 
END_VAR

// StandardPLC/Application/Global Variables/Global_Variables
VAR_GLOBAL
	
//-----------------------------------------I/O-----------------------------------------------//
	E										:INT;
	E2										:INT;
	SS										:INT;
	SS2										:INT;

//----------------------------Variables para auxilio en el primer ciclo----------------------//	
	PrimerCiclo								:BOOL := TRUE;
	gFinEncendido							:BOOL;
	TIEMPO_CICLO_DESEADO 					:UDINT := 15000;
	PosicionGrupo							:BYTE;
	gTiempoActual							:UDINT;
	gTiempoCicloMS  						:REAL;

	
//-------------------------------Variables para la cuenta atrás------------------------------//	
	SEGUNDOS_ENCENDIDO						:INT;

//-----------------------------------Entradas del sistema------------------------------------//
	gEntradasPLC							:ENTRADAS_PLC;
	gEntradasAGV							:ENTRADAS_AGV;
	
//-----------------------------------Salidas del sistema-------------------------------------//
	gSalidasPLC								:SALIDAS_PLC;

//----------------------------------Variables del variador-----------------------------------//	
	SME_DRIVER								:BOOL;
	SME_TORQUE								:INT;
	SME_SPEEDRPM_INIT						:INT;
	
	// Velocidades extension de brazo cargado
	SME_SPEEDRPM_E_Cargado_Tramo1 			:INT; 
	SME_SPEEDRPM_E_Cargado_Tramo2			:INT;
	SME_SPEEDRPM_E_Cargado_Tramo3 			:INT;
	
	// Velocidades extension de brazo descargado
	SME_SPEEDRPM_E_Descargado_Tramo1		:INT;
	SME_SPEEDRPM_E_Descargado_Tramo2		:INT;
	SME_SPEEDRPM_E_Descargado_Tramo3		:INT;
	
	// Velocidades de recoja de brazo cargado
	SME_SPEEDRPM_R_Cargado_Tramo1			:INT;
	SME_SPEEDRPM_R_Cargado_Tramo2			:INT;
	SME_SPEEDRPM_R_Cargado_Tramo3			:INT;
	
	// Velocidades de recoja de brazo descargado
	SME_SPEEDRPM_R_Descargado_Tramo2		:INT;
	SME_SPEEDRPM_R_Descargado_Tramo1		:INT;
	
	// Velocidade modo manual
	SME_SPEEDRPM_MANUAL						:INT;
	
	ConsignaA 								:INT;
	RampaTotal 								:INT;
	ConsignaVariador 						:INT;
	RampaA									:INT;
	ConsignaVariadorA						:INT;
	RestauroConsignaA 						:INT;
	RampaCumplida 							:BOOL;
	
	gRampaVelocidad							:INT;
	
	gVelocidad								:VelocidadPorTramo:=SinConsigna;
	gValorConsigna							:INT;
	gConsignaSalida							:INT;
	gEstadoRampa							:BOOL;
	gConsignaVariador						:INT;
	gConsignaA								:INT;
	gRampaTotal								:INT;
//-----------------------------------Encoder de hilo-----------------------------------------//
	Encoder									:UDINT;
	
	Recorrido_Standard						:UDINT;
	Encoder_Extendido						:UDINT;
	Encoder_Extendido_OFFSET				:UDINT;
	Encoder_Recogido_OFFSET					:UDINT;
	Encoder_Parada							:UDINT;
	TeachingOperativaB						:UDINT;

	E_Ind_Rec_MIN							:UDINT;
	E_Ind_Rec_MAX							:UDINT;
	E_Ind_Ext_MIN							:UDINT;
	E_Ind_Ext_MAX							:UDINT;
	
	Encoder_Parada_OFFSET					:UDINT;
	
	E_Anomalia_ExtenderBrazo				:UDINT;
	
	E_Tramo1								:UDINT:=0;
	E_Tramo2								:UDINT:=0;
	
	AUX_Velocidad_Inductivo					:BOOL;
	
	TeachingDone							:BOOL;
	TON_InitTeaching						:TON;
	StartCount_Encoder						:BOOL;
	gTeachingEncoder						:INT:=1;

//---------------------------------Setas de Seguridad----------------------------------------//
	RESET									:BOOL;

	HabilitarVariador						:BOOL;
	
	Setas_OPT								:INT:=1;
	
	AUX_TIMER								:BOOL;
	TON_TIMER								:TON;
	Timer_Actual_Setas						:TIME;

//------------------------------------Auxiliar Levas-----------------------------------------//	
	AUX_SubirLevas							:BOOL;
	TON_SubirLevas							:TON;
	
	AUX_BajarLevas							:BOOL;
	TON_BajarLevas							:TON;
	
	AUX_InitBajarLevas						:BOOL;
	AUX_InitSubirLevas						:BOOL;
	
	control_bajar							:INT:=1;
	control_subir							:INT:=1;

//---------------------------------------Laser-----------------------------------------------//	
	Laser 									:CamposLaser := Bumper;			
	LASER_AUX								:BOOL;
	
	AUX_LaserTimer							:BOOL;
	TON_Laser								:TON;
	AUX_Entrei:BOOL;
	Laser_OPT								:INT := 1;
	
	AccionBrazo_Laser						:INT;
	Reset_Consigna							:BOOL;
	
	AUX_SalirLaser 							:BOOL;
	TON_SalirLaser							:TON;
	Tiempo_SalidaLaser 						:TIME;

//----------------------------------AUX operativas-------------------------------------------//		
	OPT										:OperativaARealizar := indeterminado_OPT;
	OPT_Anterior 							:OperativaARealizar;
	AccionBrazo								:ControlVelocidad := A_Parar;
	gEstadoCarga							:EstadoSecuenciaCarga; 
	gEframeConCarga 						:BOOL;
	gEstadoLevas							:AccionLevas := apagado;
	gCargaOPT								:INT;
	Init_EstadoCarga						:BOOL;
	
	LevasArribaDONE							:BOOL;  //----- Variables para el control de la subida y bajada de las levas completa -----//	
	LevasAbajoDONE							:BOOL;
	
	AUX_EFrameDescargado					:BOOL; //----- Auxiliar para bajar y subir levas -----//	
	
	ParadaFotocelula						:BOOL;   //----- Variable para controlo de la subida de las levas -----//	
	
	AUX_CONT_Automatico						:INT;
	
	SetaPulsada_AUX							:BOOL;
	
	PararMotorManual						:BOOL;
	Manual_Extender							:BOOL;
	
	//----- Variables que controlan el switch...case  despues de una orden de carga o descarga -----//	
	Opt_Descarga							:INT;
	Opt_Descarga_ANT 						:INT;
	Opt_Descarga_B							:INT;
	Opt_DescargaB_ANT 						:INT;
	Opt_Carga								:INT;
	Opt_Carga_ANT 							:INT;
	OPT_Retener								:INT;
	AnchoEFrame								:INT; 
	
	AUX_DetecionCarga						:BOOL;
	TON_DetecionCarga						:TON;
	Tempo_Actual_DetecionCarga				:TIME;

//-------------------------------------AUX luces y acustico----------------------------------//		
	Disp_SelectIndicadores 					:BYTE;
	gEstadoEframe							:EstadoEframe := Identificar;    //----- Inicia el estado del E-Frame en IDENTIFICAR -----//	
	
//------------------------------------------Anomalias----------------------------------------//
	controlEstados 							:BYTE;
	PalabraAnomalia							:BYTE:= 16#FF;
	TIPO_ANOMALIA							:ARRAY[0..39] OF BYTE;
	gSupE_AnomaliasEntrada 					:ARRAY[0..39] OF BOOL :=[ 40(1)];
	
//-----------------Variables auxiliares de las anomalias del SUPERVISOR----------------------//
	gSupS_ResetExtension					:BOOL;
	gSupS_MensajeAnom						:BYTE;
	gSupS_ControlEstados					:BYTE;
	TON_Rearme								:TON;
	TOF_Rearme								:TON;
	
//-------------------Variable para saber en que estado de extension esta el brazo------------//	
	gDispS_ExtensionEstado					:BYTE;
	ParadaLaser								:BOOL := FALSE;
END_VAR

// StandardPLC/Application/CÓDIGO/PLC_PRG
PROGRAM PLC_PRG
VAR
	TiempoActualULINT		:ULINT;
	TiempoActualA			:UDINT;
	AUX_ENtrei 				:BOOL;
END_VAR

(*/////////////////////////////////////////////////////////////////////////////////////////////////////////////////////////////////////////////////////////////////////////////////////////////////////////////////////////////////////////////////////

Autor: Diana Salgado									Fecha: 17/03/2022									Versión: 35

Description:  Funcion principal 
/////////////////////////////////////////////////////////////////////////////////////////////////////////////////////////////////////////////////////////////////////////////////////////////////////////////////////////////////////////////////////*)

IN01_WIRED_INPUTS();
OUT01_WIRED_OUTPUTS();
gEntradasPLC.ModoAutomatico := E.10;

TON_Rearme(IN:=TOF_Rearme.Q, PT:=T#500MS);
TOF_Rearme(IN:=( NOT TON_Rearme.Q ), PT:=T#500MS);

//-------------------------------------------------------------------------------------------//
//-----------------------------Temporizacion para inicio de ciclo----------------------------//
//-------------------------------------------------------------------------------------------//
SysTimeGetUs(pUsTime := TiempoActualULINT);
gTiempoActual := ULINT_TO_UDINT(TiempoActualULINT);
IF NOT PrimerCiclo THEN
	gTiempoCicloMS := UDINT_TO_REAL(gTiempoActual-TiempoActualA)/1000.0;
END_IF;
TiempoActualA := gTiempoActual;

//-------------------------------------------------------------------------------------------//
//-------------------------------------Llamada a las funciones-------------------------------//
//-------------------------------------------------------------------------------------------//
IMAGENES();
SUPERVISOR();

IF PrimerCiclo THEN
	AUX_CONT_Automatico := 0;							//----- Variable para iniciar carga o descarga en modo automatico -----//
	SetaPulsada_AUX := FALSE;							//----- Variable para saber si pulsamos seta -----//
	Setas_OPT := 1;
	
	gSalidasPLC.Ch1_ReleSeguridad := TRUE;				
	gSalidasPLC.Ch2_ReleSeguridad := TRUE;				
	
	PARAMETRIZACION();
	
ELSIF (NOT PrimerCiclo) AND (NOT  SetaPulsada_AUX) THEN	
	gSalidasPLC.ContactorHabVariador 	:= TRUE;		
	
END_IF;

ESTADOS();	
Setas_Seguridad();
Laser_Seguridad();											
ACCIONES();												
SALIDAS();	
											
//-------------------------------------------------------------------------------------------//
//------------------------------Temporizacion para fin de ciclo------------------------------//
//-------------------------------------------------------------------------------------------//
TEMP00_TiempoInicio( I_TiempoEncendido:=SEGUNDOS_ENCENDIDO, O_FinTiempo=>gFinEncendido);

IF gFinEncendido THEN									//----- Cuando termina la cuenta atras, la variable PrimerCiclo es reseteada -----//
	PrimerCiclo := FALSE;
END_IF

END_PROGRAM

// StandardPLC/Application/CÓDIGO/IO/IN01_WIRED_INPUTS
PROGRAM IN01_WIRED_INPUTS
VAR
	ENTRADA0000:fb_InputAddConf_sp_ST_V02;
	ENTRADA0001:fb_InputAddConf_sp_ST_V02;
	ENTRADA0002:fb_InputAddConf_sp_ST_V02;
	ENTRADA0003:fb_InputAddConf_sp_ST_V02;
	ENTRADA0100:fb_InputAddConf_sp_ST_V02;
	ENTRADA0101:fb_InputAddConf_sp_ST_V02;
	ENTRADA0102:fb_InputAddConf_sp_ST_V02;
	ENTRADA0103:fb_InputAddConf_sp_ST_V02;
	ENTRADA0200:fb_InputAddConf_sp_ST_V02;
	ENTRADA0201:fb_InputAddConf_sp_ST_V02;
	ENTRADA0202:fb_InputAddConf_sp_ST_V02;
	ENTRADA0203:fb_InputAddConf_sp_ST_V02;
	ENTRADA0300:fb_InputAddConf_sp_ST_V02;
	ENTRADA0301:fb_InputAddConf_sp_ST_V02;
	ENTRADA0400:fb_InputAddConf_sp_ST_V02;
	ENTRADA0401:fb_InputAddConf_sp_ST_V02;
	ENTRADA0500:fb_InputAddConf_sp_ST_V02;
	ENTRADA0501:fb_InputAddConf_sp_ST_V02;
	ENTRADA0502:fb_InputAddConf_sp_ST_V02;
	ENTRADA0503:fb_InputAddConf_sp_ST_V02;
	ENTRADA0600:fb_InputAddConf_sp_ST_V02;
	ENTRADA0601:fb_InputAddConf_sp_ST_V02;
	ENTRADA0602:fb_InputAddConf_sp_ST_V02;
	ENTRADA0603:fb_InputAddConf_sp_ST_V02;
	ENTRADA0700:fb_InputAddConf_sp_ST_V02;
	ENTRADA0701:fb_InputAddConf_sp_ST_V02;
	ENTRADA0702:fb_InputAddConf_sp_ST_V02;
	ENTRADA0703:fb_InputAddConf_sp_ST_V02;
	ENTRADA0800:fb_InputAddConf_sp_ST_V02;
	ENTRADA0801:fb_InputAddConf_sp_ST_V02;
	ENTRADA0900:fb_InputAddConf_sp_ST_V02;
	ENTRADA0901:fb_InputAddConf_sp_ST_V02;
END_VAR


ENTRADA0000(IN_ResetError:=1, IN_uiChannel:=0000,IN_eModeChannel:=ifmIOcommon.MODE_INPUT.IN_DIGITAL_CSI,IN_eDestination:=ifmIOconfigDiagProt.DEST.INPUT,IN_eDiagMode:=ifmIOconfigDiagProt.eDIAG_PROT_MODE.NO_DIAG,IN_uiDetectionTime:=1000,IN_uiDiagLimMin:=0,IN_uiDiagLimMax:=2500);
ENTRADA0001(IN_ResetError:=1, IN_uiChannel:=0001,IN_eModeChannel:=ifmIOcommon.MODE_INPUT.IN_DIGITAL_CSI,IN_eDestination:=ifmIOconfigDiagProt.DEST.INPUT,IN_eDiagMode:=ifmIOconfigDiagProt.eDIAG_PROT_MODE.NO_DIAG,IN_uiDetectionTime:=1000,IN_uiDiagLimMin:=0,IN_uiDiagLimMax:=2500);
ENTRADA0002(IN_ResetError:=1, IN_uiChannel:=0002,IN_eModeChannel:=ifmIOcommon.MODE_INPUT.IN_DIGITAL_CSI,IN_eDestination:=ifmIOconfigDiagProt.DEST.INPUT,IN_eDiagMode:=ifmIOconfigDiagProt.eDIAG_PROT_MODE.NO_DIAG,IN_uiDetectionTime:=1000,IN_uiDiagLimMin:=0,IN_uiDiagLimMax:=2500);
ENTRADA0003(IN_ResetError:=1, IN_uiChannel:=0003,IN_eModeChannel:=ifmIOcommon.MODE_INPUT.IN_DIGITAL_CSI,IN_eDestination:=ifmIOconfigDiagProt.DEST.INPUT,IN_eDiagMode:=ifmIOconfigDiagProt.eDIAG_PROT_MODE.NO_DIAG,IN_uiDetectionTime:=1000,IN_uiDiagLimMin:=0,IN_uiDiagLimMax:=2500);
ENTRADA0100(IN_ResetError:=1, IN_uiChannel:=0100,IN_eModeChannel:=ifmIOcommon.MODE_INPUT.IN_DIGITAL_CSI,IN_eDestination:=ifmIOconfigDiagProt.DEST.INPUT,IN_eDiagMode:=ifmIOconfigDiagProt.eDIAG_PROT_MODE.NO_DIAG,IN_uiDetectionTime:=1000,IN_uiDiagLimMin:=0,IN_uiDiagLimMax:=2500);
ENTRADA0101(IN_ResetError:=1, IN_uiChannel:=0101,IN_eModeChannel:=ifmIOcommon.MODE_INPUT.IN_DIGITAL_CSI,IN_eDestination:=ifmIOconfigDiagProt.DEST.INPUT,IN_eDiagMode:=ifmIOconfigDiagProt.eDIAG_PROT_MODE.NO_DIAG,IN_uiDetectionTime:=1000,IN_uiDiagLimMin:=0,IN_uiDiagLimMax:=2500);
ENTRADA0102(IN_ResetError:=1, IN_uiChannel:=0102,IN_eModeChannel:=ifmIOcommon.MODE_INPUT.IN_DIGITAL_CSI,IN_eDestination:=ifmIOconfigDiagProt.DEST.INPUT,IN_eDiagMode:=ifmIOconfigDiagProt.eDIAG_PROT_MODE.NO_DIAG,IN_uiDetectionTime:=1000,IN_uiDiagLimMin:=0,IN_uiDiagLimMax:=2500);
ENTRADA0103(IN_ResetError:=1, IN_uiChannel:=0103,IN_eModeChannel:=ifmIOcommon.MODE_INPUT.IN_DIGITAL_CSI,IN_eDestination:=ifmIOconfigDiagProt.DEST.INPUT,IN_eDiagMode:=ifmIOconfigDiagProt.eDIAG_PROT_MODE.NO_DIAG,IN_uiDetectionTime:=1000,IN_uiDiagLimMin:=0,IN_uiDiagLimMax:=2500);
ENTRADA0200(IN_ResetError:=1, IN_uiChannel:=0200,IN_eModeChannel:=ifmIOcommon.MODE_INPUT.IN_DIGITAL_CSI,IN_eDestination:=ifmIOconfigDiagProt.DEST.INPUT,IN_eDiagMode:=ifmIOconfigDiagProt.eDIAG_PROT_MODE.NO_DIAG,IN_uiDetectionTime:=1000,IN_uiDiagLimMin:=0,IN_uiDiagLimMax:=2500);
ENTRADA0201(IN_ResetError:=1, IN_uiChannel:=0201,IN_eModeChannel:=ifmIOcommon.MODE_INPUT.IN_DIGITAL_CSI,IN_eDestination:=ifmIOconfigDiagProt.DEST.INPUT,IN_eDiagMode:=ifmIOconfigDiagProt.eDIAG_PROT_MODE.NO_DIAG,IN_uiDetectionTime:=1000,IN_uiDiagLimMin:=0,IN_uiDiagLimMax:=2500);
ENTRADA0202(IN_ResetError:=1, IN_uiChannel:=0202,IN_eModeChannel:=ifmIOcommon.MODE_INPUT.IN_DIGITAL_CSI,IN_eDestination:=ifmIOconfigDiagProt.DEST.INPUT,IN_eDiagMode:=ifmIOconfigDiagProt.eDIAG_PROT_MODE.NO_DIAG,IN_uiDetectionTime:=1000,IN_uiDiagLimMin:=0,IN_uiDiagLimMax:=2500);
ENTRADA0203(IN_ResetError:=1, IN_uiChannel:=0203,IN_eModeChannel:=ifmIOcommon.MODE_INPUT.IN_DIGITAL_CSI,IN_eDestination:=ifmIOconfigDiagProt.DEST.INPUT,IN_eDiagMode:=ifmIOconfigDiagProt.eDIAG_PROT_MODE.NO_DIAG,IN_uiDetectionTime:=1000,IN_uiDiagLimMin:=0,IN_uiDiagLimMax:=2500);
ENTRADA0300(IN_ResetError:=1, IN_uiChannel:=0300,IN_eModeChannel:=ifmIOcommon.MODE_INPUT.IN_DIGITAL_CSI,IN_eDestination:=ifmIOconfigDiagProt.DEST.INPUT,IN_eDiagMode:=ifmIOconfigDiagProt.eDIAG_PROT_MODE.NO_DIAG,IN_uiDetectionTime:=1000,IN_uiDiagLimMin:=0,IN_uiDiagLimMax:=2500);
ENTRADA0301(IN_ResetError:=1, IN_uiChannel:=0301,IN_eModeChannel:=ifmIOcommon.MODE_INPUT.IN_DIGITAL_CSI,IN_eDestination:=ifmIOconfigDiagProt.DEST.INPUT,IN_eDiagMode:=ifmIOconfigDiagProt.eDIAG_PROT_MODE.NO_DIAG,IN_uiDetectionTime:=1000,IN_uiDiagLimMin:=0,IN_uiDiagLimMax:=2500);
ENTRADA0400(IN_ResetError:=1, IN_uiChannel:=0400,IN_eModeChannel:=ifmIOcommon.MODE_INPUT.IN_DIGITAL_CSI,IN_eDestination:=ifmIOconfigDiagProt.DEST.INPUT,IN_eDiagMode:=ifmIOconfigDiagProt.eDIAG_PROT_MODE.NO_DIAG,IN_uiDetectionTime:=1000,IN_uiDiagLimMin:=0,IN_uiDiagLimMax:=2500);
ENTRADA0401(IN_ResetError:=1, IN_uiChannel:=0401,IN_eModeChannel:=ifmIOcommon.MODE_INPUT.IN_DIGITAL_CSI,IN_eDestination:=ifmIOconfigDiagProt.DEST.INPUT,IN_eDiagMode:=ifmIOconfigDiagProt.eDIAG_PROT_MODE.NO_DIAG,IN_uiDetectionTime:=1000,IN_uiDiagLimMin:=0,IN_uiDiagLimMax:=2500);
ENTRADA0500(IN_ResetError:=1, IN_uiChannel:=0500,IN_eModeChannel:=ifmIOcommon.MODE_INPUT.IN_DIGITAL_CSI,IN_eDestination:=ifmIOconfigDiagProt.DEST.INPUT,IN_eDiagMode:=ifmIOconfigDiagProt.eDIAG_PROT_MODE.NO_DIAG,IN_uiDetectionTime:=1000,IN_uiDiagLimMin:=0,IN_uiDiagLimMax:=2500);
ENTRADA0501(IN_ResetError:=1, IN_uiChannel:=0501,IN_eModeChannel:=ifmIOcommon.MODE_INPUT.IN_DIGITAL_CSI,IN_eDestination:=ifmIOconfigDiagProt.DEST.INPUT,IN_eDiagMode:=ifmIOconfigDiagProt.eDIAG_PROT_MODE.NO_DIAG,IN_uiDetectionTime:=1000,IN_uiDiagLimMin:=0,IN_uiDiagLimMax:=2500);
ENTRADA0502(IN_ResetError:=1, IN_uiChannel:=0502,IN_eModeChannel:=ifmIOcommon.MODE_INPUT.IN_DIGITAL_CSI,IN_eDestination:=ifmIOconfigDiagProt.DEST.INPUT,IN_eDiagMode:=ifmIOconfigDiagProt.eDIAG_PROT_MODE.NO_DIAG,IN_uiDetectionTime:=1000,IN_uiDiagLimMin:=0,IN_uiDiagLimMax:=2500);
ENTRADA0503(IN_ResetError:=1, IN_uiChannel:=0503,IN_eModeChannel:=ifmIOcommon.MODE_INPUT.IN_DIGITAL_CSI,IN_eDestination:=ifmIOconfigDiagProt.DEST.INPUT,IN_eDiagMode:=ifmIOconfigDiagProt.eDIAG_PROT_MODE.NO_DIAG,IN_uiDetectionTime:=1000,IN_uiDiagLimMin:=0,IN_uiDiagLimMax:=2500);
ENTRADA0600(IN_ResetError:=1, IN_uiChannel:=0600,IN_eModeChannel:=ifmIOcommon.MODE_INPUT.IN_DIGITAL_CSI,IN_eDestination:=ifmIOconfigDiagProt.DEST.INPUT,IN_eDiagMode:=ifmIOconfigDiagProt.eDIAG_PROT_MODE.NO_DIAG,IN_uiDetectionTime:=1000,IN_uiDiagLimMin:=0,IN_uiDiagLimMax:=2500);
ENTRADA0601(IN_ResetError:=1, IN_uiChannel:=0601,IN_eModeChannel:=ifmIOcommon.MODE_INPUT.IN_DIGITAL_CSI,IN_eDestination:=ifmIOconfigDiagProt.DEST.INPUT,IN_eDiagMode:=ifmIOconfigDiagProt.eDIAG_PROT_MODE.NO_DIAG,IN_uiDetectionTime:=1000,IN_uiDiagLimMin:=0,IN_uiDiagLimMax:=2500);
ENTRADA0602(IN_ResetError:=1, IN_uiChannel:=0602,IN_eModeChannel:=ifmIOcommon.MODE_INPUT.IN_DIGITAL_CSI,IN_eDestination:=ifmIOconfigDiagProt.DEST.INPUT,IN_eDiagMode:=ifmIOconfigDiagProt.eDIAG_PROT_MODE.NO_DIAG,IN_uiDetectionTime:=1000,IN_uiDiagLimMin:=0,IN_uiDiagLimMax:=2500);
ENTRADA0603(IN_ResetError:=1, IN_uiChannel:=0603,IN_eModeChannel:=ifmIOcommon.MODE_INPUT.IN_DIGITAL_CSI,IN_eDestination:=ifmIOconfigDiagProt.DEST.INPUT,IN_eDiagMode:=ifmIOconfigDiagProt.eDIAG_PROT_MODE.NO_DIAG,IN_uiDetectionTime:=1000,IN_uiDiagLimMin:=0,IN_uiDiagLimMax:=2500);
ENTRADA0700(IN_ResetError:=1, IN_uiChannel:=0700,IN_eModeChannel:=ifmIOcommon.MODE_INPUT.IN_DIGITAL_CSI,IN_eDestination:=ifmIOconfigDiagProt.DEST.INPUT,IN_eDiagMode:=ifmIOconfigDiagProt.eDIAG_PROT_MODE.NO_DIAG,IN_uiDetectionTime:=1000,IN_uiDiagLimMin:=0,IN_uiDiagLimMax:=2500);
ENTRADA0701(IN_ResetError:=1, IN_uiChannel:=0701,IN_eModeChannel:=ifmIOcommon.MODE_INPUT.IN_DIGITAL_CSI,IN_eDestination:=ifmIOconfigDiagProt.DEST.INPUT,IN_eDiagMode:=ifmIOconfigDiagProt.eDIAG_PROT_MODE.NO_DIAG,IN_uiDetectionTime:=1000,IN_uiDiagLimMin:=0,IN_uiDiagLimMax:=2500);
ENTRADA0702(IN_ResetError:=1, IN_uiChannel:=0702,IN_eModeChannel:=ifmIOcommon.MODE_INPUT.IN_DIGITAL_CSI,IN_eDestination:=ifmIOconfigDiagProt.DEST.INPUT,IN_eDiagMode:=ifmIOconfigDiagProt.eDIAG_PROT_MODE.NO_DIAG,IN_uiDetectionTime:=1000,IN_uiDiagLimMin:=0,IN_uiDiagLimMax:=2500);
ENTRADA0703(IN_ResetError:=1, IN_uiChannel:=0703,IN_eModeChannel:=ifmIOcommon.MODE_INPUT.IN_DIGITAL_CSI,IN_eDestination:=ifmIOconfigDiagProt.DEST.INPUT,IN_eDiagMode:=ifmIOconfigDiagProt.eDIAG_PROT_MODE.NO_DIAG,IN_uiDetectionTime:=1000,IN_uiDiagLimMin:=0,IN_uiDiagLimMax:=2500);
ENTRADA0800(IN_ResetError:=1, IN_uiChannel:=0800,IN_eModeChannel:=ifmIOcommon.MODE_INPUT.IN_DIGITAL_CSI,IN_eDestination:=ifmIOconfigDiagProt.DEST.INPUT,IN_eDiagMode:=ifmIOconfigDiagProt.eDIAG_PROT_MODE.NO_DIAG,IN_uiDetectionTime:=1000,IN_uiDiagLimMin:=0,IN_uiDiagLimMax:=2500);
ENTRADA0801(IN_ResetError:=1, IN_uiChannel:=0801,IN_eModeChannel:=ifmIOcommon.MODE_INPUT.IN_DIGITAL_CSI,IN_eDestination:=ifmIOconfigDiagProt.DEST.INPUT,IN_eDiagMode:=ifmIOconfigDiagProt.eDIAG_PROT_MODE.NO_DIAG,IN_uiDetectionTime:=1000,IN_uiDiagLimMin:=0,IN_uiDiagLimMax:=2500);
ENTRADA0900(IN_ResetError:=1, IN_uiChannel:=0900,IN_eModeChannel:=ifmIOcommon.MODE_INPUT.IN_DIGITAL_CSI,IN_eDestination:=ifmIOconfigDiagProt.DEST.INPUT,IN_eDiagMode:=ifmIOconfigDiagProt.eDIAG_PROT_MODE.NO_DIAG,IN_uiDetectionTime:=1000,IN_uiDiagLimMin:=0,IN_uiDiagLimMax:=2500);
ENTRADA0901(IN_ResetError:=1, IN_uiChannel:=0901,IN_eModeChannel:=ifmIOcommon.MODE_INPUT.IN_DIGITAL_CSI,IN_eDestination:=ifmIOconfigDiagProt.DEST.INPUT,IN_eDiagMode:=ifmIOconfigDiagProt.eDIAG_PROT_MODE.NO_DIAG,IN_uiDetectionTime:=1000,IN_uiDiagLimMin:=0,IN_uiDiagLimMax:=2500);

E.0:=ENTRADA0000.OUT_ValueDigital;
E.1:=ENTRADA0001.OUT_ValueDigital;
E.2:=ENTRADA0002.OUT_ValueDigital;
E.3:=ENTRADA0003.OUT_ValueDigital;
E.4:=ENTRADA0100.OUT_ValueDigital;
E.5:=ENTRADA0101.OUT_ValueDigital;
E.6:=ENTRADA0102.OUT_ValueDigital;
E.7:=ENTRADA0103.OUT_ValueDigital;
E.8:=ENTRADA0200.OUT_ValueDigital;
E.9:=ENTRADA0201.OUT_ValueDigital;
E.10:=ENTRADA0202.OUT_ValueDigital;
E.11:=ENTRADA0203.OUT_ValueDigital;
E.12:=ENTRADA0300.OUT_ValueDigital;
E.13:=ENTRADA0301.OUT_ValueDigital;
E.14:=ENTRADA0400.OUT_ValueDigital;
E.15:=ENTRADA0401.OUT_ValueDigital;
E2.0:=ENTRADA0500.OUT_ValueDigital;
E2.1:=ENTRADA0501.OUT_ValueDigital;
E2.2:=ENTRADA0502.OUT_ValueDigital;	
E2.3:=ENTRADA0503.OUT_ValueDigital;	
E2.4:=ENTRADA0600.OUT_ValueDigital;			//Entrada 55 - Botón brazo adelante
E2.5:=ENTRADA0601.OUT_ValueDigital;			//Entrada 56 - Botón brazo retroceso
E2.6:=ENTRADA0602.OUT_ValueDigital;	
E2.7:=ENTRADA0603.OUT_ValueDigital;	
E2.8:=ENTRADA0700.OUT_ValueDigital;	
E2.9:=ENTRADA0701.OUT_ValueDigital;	
E2.10:=ENTRADA0702.OUT_ValueDigital;	
E2.11:=ENTRADA0703.OUT_ValueDigital;	
E2.12:=ENTRADA0800.OUT_ValueDigital;
E2.13:=ENTRADA0801.OUT_ValueDigital;
E2.14:=ENTRADA0900.OUT_ValueDigital;
E2.15:=ENTRADA0901.OUT_ValueDigital;

END_PROGRAM

// StandardPLC/Application/CÓDIGO/AUX_IFM/fb_InputAddConf_sp_ST_V02
FUNCTION_BLOCK fb_InputAddConf_sp_ST_V02

VAR_INPUT
	IN_ResetError:BOOL;	
	IN_uiChannel:UINT;
	IN_eModeChannel:ifmIOcommon.MODE_INPUT;
	IN_eDestination:ifmIOconfigDiagProt.DEST;
	IN_eDiagMode:ifmIOconfigDiagProt.eDIAG_PROT_MODE;
	IN_uiDetectionTime:UINT;
	IN_uiDiagLimMin:UINT;
	IN_uiDiagLimMax:UINT;
END_VAR	
	
VAR_OUTPUT
	OUT_Done:BOOL;
	OUT_Error:BOOL;
	OUT_DiagInfo:ifmTypes.DIAG_INFO;	
	OUT_DiagInfoProt: ifmTypes.DIAG_INFO;
	OUT_DiagInfoLevel: ifmTypes.DIAG_INFO;	
	OUT_ValueDigital:BOOL;
	OUT_ValueAnalogue:UINT;
END_VAR

VAR
	
	l_xExecute:BOOL;
	ConfigDiagLevel: ifmIOconfigDiagProt.ConfigDiagLevel;
	ConfigDiagProt: ifmIOconfigDiagProt.ConfigDiagProt;
	(*ConfigSwThreshold: ifmConfigSwThreshold.ConfigSwThreshold;*)

	l_xExecute_DiagLevel:BOOL;
	l_xExecuted_DiagLevel:BOOL;	
	l_xExecute_DiagProt:BOOL;
	l_xExecuted_DiagProt:BOOL;
	l_xExecute_SwThreshold:BOOL;
	l_xExecuted_SwThreshold:BOOL;	
	R_TRIG_Execute: R_TRIG;
	Input: ifmIOcommon.Input;
	
	R_TRIG_Done: R_TRIG;
	
END_VAR
VAR // added by the converter: edge detectors and wires of the graphical bodies
    _w1 : BOOL;
END_VAR

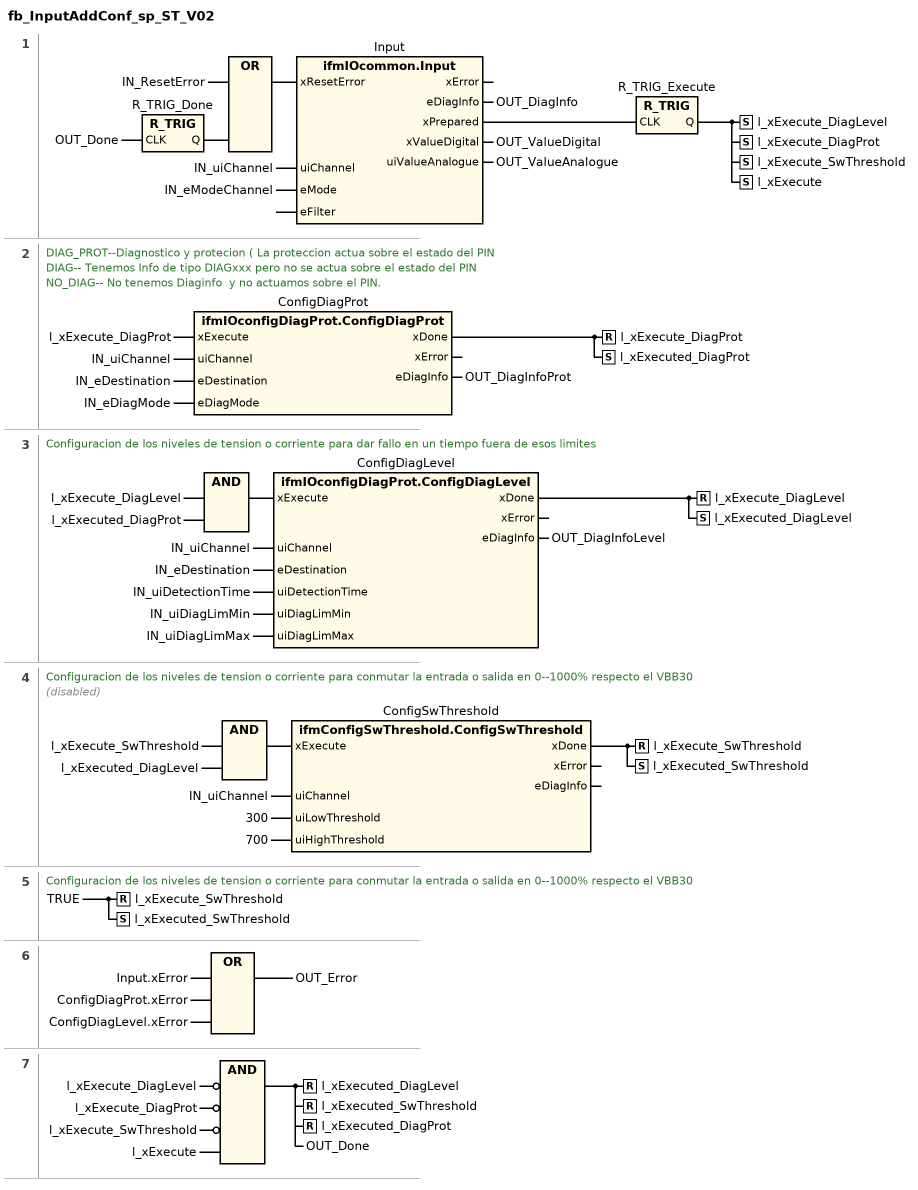
// NETWORK 1
R_TRIG_Done(CLK := OUT_Done); // R_TRIG
Input(
    xResetError := IN_ResetError OR R_TRIG_Done.Q,
    uiChannel := IN_uiChannel,
    eMode := IN_eModeChannel,
    eDiagInfo => OUT_DiagInfo,
    xValueDigital => OUT_ValueDigital,
    uiValueAnalogue => OUT_ValueAnalogue); // ifmIOcommon.Input
R_TRIG_Execute(CLK := Input.xPrepared); // R_TRIG
l_xExecute_DiagLevel S= R_TRIG_Execute.Q;
l_xExecute_DiagProt S= R_TRIG_Execute.Q;
l_xExecute_SwThreshold S= R_TRIG_Execute.Q;
l_xExecute S= R_TRIG_Execute.Q;

// NETWORK 2
// DIAG_PROT--Diagnostico y protecion ( La proteccion actua sobre el estado del PIN
// DIAG-- Tenemos Info de tipo DIAGxxx pero no se actua sobre el estado del PIN
// NO_DIAG-- No tenemos Diaginfo  y no actuamos sobre el PIN.
ConfigDiagProt(
    xExecute := l_xExecute_DiagProt,
    uiChannel := IN_uiChannel,
    eDestination := IN_eDestination,
    eDiagMode := IN_eDiagMode,
    eDiagInfo => OUT_DiagInfoProt); // ifmIOconfigDiagProt.ConfigDiagProt
l_xExecute_DiagProt R= ConfigDiagProt.xDone;
l_xExecuted_DiagProt S= ConfigDiagProt.xDone;

// NETWORK 3
// Configuracion de los niveles de tension o corriente para dar fallo en un tiempo fuera de esos limites
ConfigDiagLevel(
    xExecute := l_xExecute_DiagLevel AND l_xExecuted_DiagProt,
    uiChannel := IN_uiChannel,
    eDestination := IN_eDestination,
    uiDetectionTime := IN_uiDetectionTime,
    uiDiagLimMin := IN_uiDiagLimMin,
    uiDiagLimMax := IN_uiDiagLimMax,
    eDiagInfo => OUT_DiagInfoLevel); // ifmIOconfigDiagProt.ConfigDiagLevel
l_xExecute_DiagLevel R= ConfigDiagLevel.xDone;
l_xExecuted_DiagLevel S= ConfigDiagLevel.xDone;

// NETWORK 4 (disabled)
// Configuracion de los niveles de tension o corriente para conmutar la entrada o salida en 0--1000% respecto el VBB30
// ConfigSwThreshold(
//     xExecute := l_xExecute_SwThreshold AND l_xExecuted_DiagLevel,
//     uiChannel := IN_uiChannel,
//     uiLowThreshold := 300,
//     uiHighThreshold := 700); // ifmConfigSwThreshold.ConfigSwThreshold
// l_xExecute_SwThreshold R= ConfigSwThreshold.xDone;
// l_xExecuted_SwThreshold S= ConfigSwThreshold.xDone;

// NETWORK 5
// Configuracion de los niveles de tension o corriente para conmutar la entrada o salida en 0--1000% respecto el VBB30
l_xExecute_SwThreshold R= TRUE;
l_xExecuted_SwThreshold S= TRUE;

// NETWORK 6
OUT_Error := Input.xError OR ConfigDiagProt.xError OR ConfigDiagLevel.xError;

// NETWORK 7
_w1 := NOT l_xExecute_DiagLevel AND NOT l_xExecute_DiagProt AND NOT l_xExecute_SwThreshold AND l_xExecute;
l_xExecuted_DiagLevel R= _w1;
l_xExecuted_SwThreshold R= _w1;
l_xExecuted_DiagProt R= _w1;
OUT_Done := _w1;

END_FUNCTION_BLOCK

// StandardPLC/Application/CÓDIGO/IO/OUT01_WIRED_OUTPUTS
PROGRAM OUT01_WIRED_OUTPUTS
VAR
	GRUPO_SALIDAS0: fb_OutputGroupAddConf_sp_ST_V02;
	GRUPO_SALIDAS1: fb_OutputGroupAddConf_sp_ST_V02;
	GRUPO_SALIDAS2: fb_OutputGroupAddConf_sp_ST_V02;
	GRUPO_SALIDAS3: fb_OutputGroupAddConf_sp_ST_V02;
	SALIDA0000: fb_OutputAddConf_sp_ST_V02;
	SALIDA0001: fb_OutputAddConf_sp_ST_V02;
	SALIDA0002: fb_OutputAddConf_sp_ST_V02;
	SALIDA0003: fb_OutputAddConf_sp_ST_V02;
	SALIDA0004: fb_OutputAddConf_sp_ST_V02;
	SALIDA0005:	fb_OutputAddConf_sp_ST_V02;
	SALIDA0006:	fb_OutputAddConf_sp_ST_V02;
	SALIDAPWM0106: ifmOutPWM.PWM1000;
	(*SALIDA0006: fb_OutputAddConf_sp_ST_V02;*)
	SALIDA0007: fb_OutputAddConf_sp_ST_V02;
	SALIDA0008: fb_OutputAddConf_sp_ST_V02;
	SALIDA0100: fb_OutputAddConf_sp_ST_V02;
	SALIDA0101: fb_OutputAddConf_sp_ST_V02;
	SALIDA0102: fb_OutputAddConf_sp_ST_V02;
	SALIDA0103: fb_OutputAddConf_sp_ST_V02;
	SALIDA0104: fb_OutputAddConf_sp_ST_V02;
	SALIDA0105: fb_OutputAddConf_sp_ST_V02;
	(*SALIDAHB0106:fb_OutBridgeAddConf_sp_ST_V02;*)
	SALIDA0106: fb_OutputAddConf_sp_ST_V02;
	SALIDA0107: fb_OutputAddConf_sp_ST_V02;
	SALIDA0108: fb_OutputAddConf_sp_ST_V02;
	SALIDA0200: fb_OutputAddConf_sp_ST_V02;
	SALIDA0201: fb_OutputAddConf_sp_ST_V02;
	SALIDA0202: fb_OutputAddConf_sp_ST_V02;
	SALIDA0203: fb_OutputAddConf_sp_ST_V02;
	SALIDA0204: fb_OutputAddConf_sp_ST_V02;
	SALIDA0205: fb_OutputAddConf_sp_ST_V02;
	SALIDA0206: fb_OutputAddConf_sp_ST_V02;
	//SALIDAPWM0206: ifmOutPWM.PWM1000;
	(*SALIDA0206: fb_OutputAddConf_sp_ST_V02;*)
	SALIDA0207: fb_OutputAddConf_sp_ST_V02;
	SALIDA0208: fb_OutputAddConf_sp_ST_V02;
	SALIDA0300: fb_OutputAddConf_sp_ST_V02;
	SALIDA0301: fb_OutputAddConf_sp_ST_V02;
END_VAR


(*Activación de cada grupo de salidas*)
GRUPO_SALIDAS0(IN_ResetError:=1,IN_uiChannel:=0,IN_eModeChannel:=ifmOutGroup.MODE_OUTPUT_GROUP.OUT_DIGITAL,IN_eDestination:=ifmIOconfigDiagProt.DEST.OUT_GROUP,IN_eDiagMode:=ifmIOconfigDiagProt.eDIAG_PROT_MODE.NO_DIAG, IN_DetectionTime:=1000,IN_DiagLimMin:=0,IN_DiagLimMax:=12000,IN_Value:=1);
GRUPO_SALIDAS1(IN_ResetError:=1,IN_uiChannel:=1,IN_eModeChannel:=ifmOutGroup.MODE_OUTPUT_GROUP.OUT_DIGITAL,IN_eDestination:=ifmIOconfigDiagProt.DEST.OUT_GROUP,IN_eDiagMode:=ifmIOconfigDiagProt.eDIAG_PROT_MODE.NO_DIAG, IN_DetectionTime:=1000,IN_DiagLimMin:=0,IN_DiagLimMax:=12000,IN_Value:=1);
GRUPO_SALIDAS2(IN_ResetError:=1,IN_uiChannel:=2,IN_eModeChannel:=ifmOutGroup.MODE_OUTPUT_GROUP.OUT_DIGITAL,IN_eDestination:=ifmIOconfigDiagProt.DEST.OUT_GROUP,IN_eDiagMode:=ifmIOconfigDiagProt.eDIAG_PROT_MODE.NO_DIAG, IN_DetectionTime:=1000,IN_DiagLimMin:=0,IN_DiagLimMax:=12000,IN_Value:=1);
GRUPO_SALIDAS3(IN_ResetError:=1,IN_uiChannel:=3,IN_eModeChannel:=ifmOutGroup.MODE_OUTPUT_GROUP.OUT_DIGITAL,IN_eDestination:=ifmIOconfigDiagProt.DEST.OUT_GROUP,IN_eDiagMode:=ifmIOconfigDiagProt.eDIAG_PROT_MODE.NO_DIAG, IN_DetectionTime:=1000,IN_DiagLimMin:=0,IN_DiagLimMax:=12000,IN_Value:=1);

(*Valor salidas*)
SALIDA0000(IN_ResetError:=1,IN_uiChannel:=0000,IN_eModeChannel:=ifmIOCommon.MODE_OUTPUT.OUT_DIGITAL_CSO,IN_eDestination:=ifmIOconfigDiagProt.DEST.OUTPUT,IN_eDiagMode:=ifmIOconfigDiagProt.eDIAG_PROT_MODE.NO_DIAG, IN_DetectionTime:=1000,IN_DiagLimMin:=0,IN_DiagLimMax:=2500,IN_Value:=SS.0);
SALIDA0001(IN_ResetError:=1,IN_uiChannel:=0001,IN_eModeChannel:=ifmIOCommon.MODE_OUTPUT.OUT_DIGITAL_CSO,IN_eDestination:=ifmIOconfigDiagProt.DEST.OUTPUT,IN_eDiagMode:=ifmIOconfigDiagProt.eDIAG_PROT_MODE.NO_DIAG, IN_DetectionTime:=1000,IN_DiagLimMin:=0,IN_DiagLimMax:=2500,IN_Value:=SS.1);
SALIDA0002(IN_ResetError:=1,IN_uiChannel:=0002,IN_eModeChannel:=ifmIOCommon.MODE_OUTPUT.OUT_DIGITAL_CSO,IN_eDestination:=ifmIOconfigDiagProt.DEST.OUTPUT,IN_eDiagMode:=ifmIOconfigDiagProt.eDIAG_PROT_MODE.NO_DIAG, IN_DetectionTime:=1000,IN_DiagLimMin:=0,IN_DiagLimMax:=2500,IN_Value:=SS.2);
SALIDA0003(IN_ResetError:=1,IN_uiChannel:=0003,IN_eModeChannel:=ifmIOCommon.MODE_OUTPUT.OUT_DIGITAL_CSO,IN_eDestination:=ifmIOconfigDiagProt.DEST.OUTPUT,IN_eDiagMode:=ifmIOconfigDiagProt.eDIAG_PROT_MODE.NO_DIAG, IN_DetectionTime:=1000,IN_DiagLimMin:=0,IN_DiagLimMax:=2500,IN_Value:=SS.3);
SALIDA0004(IN_ResetError:=1,IN_uiChannel:=0004,IN_eModeChannel:=ifmIOCommon.MODE_OUTPUT.OUT_DIGITAL_CSO,IN_eDestination:=ifmIOconfigDiagProt.DEST.OUTPUT,IN_eDiagMode:=ifmIOconfigDiagProt.eDIAG_PROT_MODE.NO_DIAG, IN_DetectionTime:=1000,IN_DiagLimMin:=0,IN_DiagLimMax:=2500,IN_Value:=SS.4);
SALIDA0005(IN_ResetError:=1,IN_uiChannel:=0005,IN_eModeChannel:=ifmIOCommon.MODE_OUTPUT.OUT_DIGITAL_CSO,IN_eDestination:=ifmIOconfigDiagProt.DEST.OUTPUT,IN_eDiagMode:=ifmIOconfigDiagProt.eDIAG_PROT_MODE.NO_DIAG, IN_DetectionTime:=1000,IN_DiagLimMin:=0,IN_DiagLimMax:=2500,IN_Value:=SS.5);	
SALIDA0006(IN_ResetError:=1,IN_uiChannel:=0006,IN_eModeChannel:=ifmIOCommon.MODE_OUTPUT.OUT_DIGITAL_CSO,IN_eDestination:=ifmIOconfigDiagProt.DEST.OUTPUT,IN_eDiagMode:=ifmIOconfigDiagProt.eDIAG_PROT_MODE.NO_DIAG, IN_DetectionTime:=1000,IN_DiagLimMin:=0,IN_DiagLimMax:=2500,IN_Value:=SS.6);
SALIDA0007(IN_ResetError:=1,IN_uiChannel:=0007,IN_eModeChannel:=ifmIOCommon.MODE_OUTPUT.OUT_DIGITAL_CSO,IN_eDestination:=ifmIOconfigDiagProt.DEST.OUTPUT,IN_eDiagMode:=ifmIOconfigDiagProt.eDIAG_PROT_MODE.NO_DIAG, IN_DetectionTime:=1000,IN_DiagLimMin:=0,IN_DiagLimMax:=2500,IN_Value:=SS.7);
SALIDA0008(IN_ResetError:=1,IN_uiChannel:=0008,IN_eModeChannel:=ifmIOCommon.MODE_OUTPUT.OUT_DIGITAL_CSO,IN_eDestination:=ifmIOconfigDiagProt.DEST.OUTPUT,IN_eDiagMode:=ifmIOconfigDiagProt.eDIAG_PROT_MODE.NO_DIAG, IN_DetectionTime:=1000,IN_DiagLimMin:=0,IN_DiagLimMax:=2500,IN_Value:=SS.8);
SALIDA0100(IN_ResetError:=1,IN_uiChannel:=0100,IN_eModeChannel:=ifmIOCommon.MODE_OUTPUT.OUT_DIGITAL_CSO,IN_eDestination:=ifmIOconfigDiagProt.DEST.OUTPUT,IN_eDiagMode:=ifmIOconfigDiagProt.eDIAG_PROT_MODE.NO_DIAG, IN_DetectionTime:=1000,IN_DiagLimMin:=0,IN_DiagLimMax:=2500,IN_Value:=SS.9);

SALIDA0101(IN_ResetError:=1,IN_uiChannel:=0101,IN_eModeChannel:=ifmIOCommon.MODE_OUTPUT.OUT_DIGITAL_CSO,IN_eDestination:=ifmIOconfigDiagProt.DEST.OUTPUT,IN_eDiagMode:=ifmIOconfigDiagProt.eDIAG_PROT_MODE.NO_DIAG, IN_DetectionTime:=1000,IN_DiagLimMin:=0,IN_DiagLimMax:=2500,IN_Value:=SS.10);
SALIDA0102(IN_ResetError:=1,IN_uiChannel:=0102,IN_eModeChannel:=ifmIOCommon.MODE_OUTPUT.OUT_DIGITAL_CSO,IN_eDestination:=ifmIOconfigDiagProt.DEST.OUTPUT,IN_eDiagMode:=ifmIOconfigDiagProt.eDIAG_PROT_MODE.NO_DIAG, IN_DetectionTime:=1000,IN_DiagLimMin:=0,IN_DiagLimMax:=2500,IN_Value:=SS.11);
SALIDA0103(IN_ResetError:=1,IN_uiChannel:=0103,IN_eModeChannel:=ifmIOCommon.MODE_OUTPUT.OUT_DIGITAL_CSO,IN_eDestination:=ifmIOconfigDiagProt.DEST.OUTPUT,IN_eDiagMode:=ifmIOconfigDiagProt.eDIAG_PROT_MODE.NO_DIAG, IN_DetectionTime:=1000,IN_DiagLimMin:=0,IN_DiagLimMax:=2500,IN_Value:=SS.12);
SALIDA0104(IN_ResetError:=1,IN_uiChannel:=0104,IN_eModeChannel:=ifmIOCommon.MODE_OUTPUT.OUT_DIGITAL_CSO,IN_eDestination:=ifmIOconfigDiagProt.DEST.OUTPUT,IN_eDiagMode:=ifmIOconfigDiagProt.eDIAG_PROT_MODE.NO_DIAG, IN_DetectionTime:=1000,IN_DiagLimMin:=0,IN_DiagLimMax:=2500,IN_Value:=SS.13);
SALIDA0105(IN_ResetError:=1,IN_uiChannel:=0105,IN_eModeChannel:=ifmIOCommon.MODE_OUTPUT.OUT_DIGITAL_CSO,IN_eDestination:=ifmIOconfigDiagProt.DEST.OUTPUT,IN_eDiagMode:=ifmIOconfigDiagProt.eDIAG_PROT_MODE.NO_DIAG, IN_DetectionTime:=1000,IN_DiagLimMin:=0,IN_DiagLimMax:=2500,IN_Value:=SS.14);
SALIDAPWM0106(uiChannel := 106, eMode := ifmOutPWM.MODE_PWM.OUT_PWM_CSO, uiFrequency := 250, uiValue := BOOL_TO_UINT(SS.15)*1000, uiDitherFrequency:= 0, uiDitherValue:= 0);
SALIDA0107(IN_ResetError:=1,IN_uiChannel:=0107,IN_eModeChannel:=ifmIOCommon.MODE_OUTPUT.OUT_DIGITAL_CSO,IN_eDestination:=ifmIOconfigDiagProt.DEST.OUTPUT,IN_eDiagMode:=ifmIOconfigDiagProt.eDIAG_PROT_MODE.NO_DIAG, IN_DetectionTime:=1000,IN_DiagLimMin:=0,IN_DiagLimMax:=2500,IN_Value:=SS2.0);
SALIDA0108(IN_ResetError:=1,IN_uiChannel:=0108,IN_eModeChannel:=ifmIOCommon.MODE_OUTPUT.OUT_DIGITAL_CSO,IN_eDestination:=ifmIOconfigDiagProt.DEST.OUTPUT,IN_eDiagMode:=ifmIOconfigDiagProt.eDIAG_PROT_MODE.NO_DIAG, IN_DetectionTime:=1000,IN_DiagLimMin:=0,IN_DiagLimMax:=4500,IN_Value:=SS2.1);
SALIDA0200(IN_ResetError:=1,IN_uiChannel:=0200,IN_eModeChannel:=ifmIOCommon.MODE_OUTPUT.OUT_DIGITAL_CSO,IN_eDestination:=ifmIOconfigDiagProt.DEST.OUTPUT,IN_eDiagMode:=ifmIOconfigDiagProt.eDIAG_PROT_MODE.NO_DIAG, IN_DetectionTime:=1000,IN_DiagLimMin:=0,IN_DiagLimMax:=2500,IN_Value:=SS2.2);
SALIDA0201(IN_ResetError:=1,IN_uiChannel:=0201,IN_eModeChannel:=ifmIOCommon.MODE_OUTPUT.OUT_DIGITAL_CSO,IN_eDestination:=ifmIOconfigDiagProt.DEST.OUTPUT,IN_eDiagMode:=ifmIOconfigDiagProt.eDIAG_PROT_MODE.NO_DIAG, IN_DetectionTime:=1000,IN_DiagLimMin:=0,IN_DiagLimMax:=2500,IN_Value:=SS2.3);
SALIDA0202(IN_ResetError:=1,IN_uiChannel:=0202,IN_eModeChannel:=ifmIOCommon.MODE_OUTPUT.OUT_DIGITAL_CSO,IN_eDestination:=ifmIOconfigDiagProt.DEST.OUTPUT,IN_eDiagMode:=ifmIOconfigDiagProt.eDIAG_PROT_MODE.NO_DIAG, IN_DetectionTime:=1000,IN_DiagLimMin:=0,IN_DiagLimMax:=2500,IN_Value:=SS2.4);
SALIDA0203(IN_ResetError:=1,IN_uiChannel:=0203,IN_eModeChannel:=ifmIOCommon.MODE_OUTPUT.OUT_DIGITAL_CSO,IN_eDestination:=ifmIOconfigDiagProt.DEST.OUTPUT,IN_eDiagMode:=ifmIOconfigDiagProt.eDIAG_PROT_MODE.NO_DIAG, IN_DetectionTime:=1000,IN_DiagLimMin:=0,IN_DiagLimMax:=2500,IN_Value:=SS2.5);
SALIDA0204(IN_ResetError:=1,IN_uiChannel:=0204,IN_eModeChannel:=ifmIOCommon.MODE_OUTPUT.OUT_DIGITAL_CSO,IN_eDestination:=ifmIOconfigDiagProt.DEST.OUTPUT,IN_eDiagMode:=ifmIOconfigDiagProt.eDIAG_PROT_MODE.NO_DIAG, IN_DetectionTime:=1000,IN_DiagLimMin:=0,IN_DiagLimMax:=2500,IN_Value:=SS2.6);
SALIDA0205(IN_ResetError:=1,IN_uiChannel:=0205,IN_eModeChannel:=ifmIOCommon.MODE_OUTPUT.OUT_DIGITAL_CSO,IN_eDestination:=ifmIOconfigDiagProt.DEST.OUTPUT,IN_eDiagMode:=ifmIOconfigDiagProt.eDIAG_PROT_MODE.NO_DIAG, IN_DetectionTime:=1000,IN_DiagLimMin:=0,IN_DiagLimMax:=2500,IN_Value:=SS2.7);
SALIDA0206(IN_ResetError:=1,IN_uiChannel:=0206,IN_eModeChannel:=ifmIOCommon.MODE_OUTPUT.OUT_DIGITAL_CSO,IN_eDestination:=ifmIOconfigDiagProt.DEST.OUTPUT,IN_eDiagMode:=ifmIOconfigDiagProt.eDIAG_PROT_MODE.NO_DIAG, IN_DetectionTime:=1000,IN_DiagLimMin:=0,IN_DiagLimMax:=2500,IN_Value:=SS2.8);


//SALIDAPWM0206(uiChannel := 206, eMode := ifmOutPWM.MODE_PWM.OUT_PWM_CSO, uiFrequency := 250, uiValue := BOOL_TO_UINT(SS2.8)*1000, uiDitherFrequency:= 0, uiDitherValue:= 0);		
SALIDA0207(IN_ResetError:=1,IN_uiChannel:=0207,IN_eModeChannel:=ifmIOCommon.MODE_OUTPUT.OUT_DIGITAL_CSO,IN_eDestination:=ifmIOconfigDiagProt.DEST.OUTPUT,IN_eDiagMode:=ifmIOconfigDiagProt.eDIAG_PROT_MODE.NO_DIAG, IN_DetectionTime:=1000,IN_DiagLimMin:=0,IN_DiagLimMax:=2500,IN_Value:=SS2.9);
SALIDA0208(IN_ResetError:=1,IN_uiChannel:=0208,IN_eModeChannel:=ifmIOCommon.MODE_OUTPUT.OUT_DIGITAL_CSO,IN_eDestination:=ifmIOconfigDiagProt.DEST.OUTPUT,IN_eDiagMode:=ifmIOconfigDiagProt.eDIAG_PROT_MODE.NO_DIAG, IN_DetectionTime:=1000,IN_DiagLimMin:=0,IN_DiagLimMax:=2500,IN_Value:=SS2.10);
SALIDA0300(IN_ResetError:=1,IN_uiChannel:=0300,IN_eModeChannel:=ifmIOCommon.MODE_OUTPUT.OUT_DIGITAL_CSO,IN_eDestination:=ifmIOconfigDiagProt.DEST.OUTPUT,IN_eDiagMode:=ifmIOconfigDiagProt.eDIAG_PROT_MODE.NO_DIAG, IN_DetectionTime:=1000,IN_DiagLimMin:=0,IN_DiagLimMax:=2500,IN_Value:=SS2.11);
SALIDA0301(IN_ResetError:=1,IN_uiChannel:=0301,IN_eModeChannel:=ifmIOCommon.MODE_OUTPUT.OUT_DIGITAL_CSO,IN_eDestination:=ifmIOconfigDiagProt.DEST.OUTPUT,IN_eDiagMode:=ifmIOconfigDiagProt.eDIAG_PROT_MODE.NO_DIAG, IN_DetectionTime:=1000,IN_DiagLimMin:=0,IN_DiagLimMax:=2500,IN_Value:=SS2.12);

END_PROGRAM

// StandardPLC/Application/CÓDIGO/SALIDAS
PROGRAM SALIDAS
VAR
	estadoEframe 				:BYTE;

	TON_InitializacionSME		:TON;
	TON_Reposo					:TON;
	
	AuxRampaLaser				:BOOL;
	
	
	// Variables Encoder
	AUX							:INT:=1;
	
	CAN_ENABLE					:ifmRCAN.CAN_Enable;
	
	Encoder_inicial				:UDINT;
	
	TON1 						:TON;
	
	MatrizEnvio1				: ARRAY[0..7] OF USINT;
	MatrizEnvio2				: ARRAY[0..7] OF USINT;
	
	CAN_TX1						:ifmRCAN.CAN_Tx;
	CAN_TX2						:ifmRCAN.CAN_Tx;
END_VAR

(*/////////////////////////////////////////////////////////////////////////////////////////////////////////////////////////////////////////////////////////////////////////////////////////////////////////////////////////////////////////////////////
SALIDAS (PRG)                     

Description:  Módulo encargado de mapear salidas
			 
///////////////////////////////////////////////////////////////////////////////////////////////////////////////////////////////////////////////////////////////////////////////////////////////////////////////////////////////////////////////////// *)

//-------------------------------------------------------------------------------------------//
//----------------------------------Salidas del PLC cableadas--------------------------------//
//-------------------------------------------------------------------------------------------//
OUT01_WIRED_OUTPUTS();

SS2.5 	:= 	gSalidasPLC.LuzAmarillo;
SS2.3	:=	gSalidasPLC.LuzRojo;.
SS2.4 	:=  gSalidasPLC.LuzVerde;
SS2.2   :=  gSalidasPLC.Acustico;
SS2.6	:=	gSalidasPLC.LuzBotonRearme;

SS2.0 := gSalidasPLC.SubirLevas;
SS2.1 := gSalidasPLC.BajarLevas;

SS.1	:= gSalidasPLC.Contactor; 
SS.10	:= gSalidasPLC.Contactor2;

SS2.8	:= gSalidasPLC.Eletrofreno;

SS2.7	:= gSalidasPLC.ContactorHabVariador;

SS.7	:= gSalidasPLC.SetaEmergenciaOUT1;
SS.8	:= gSalidasPLC.SetaEmergenciaOUT2;

SS.5 := gSalidasPLC.Ch1_ReleSeguridad;
SS.14 := gSalidasPLC.Ch2_ReleSeguridad;

Campos_Laser();
SS.2 := gSalidasPLC.LaserA;
SS.3 := gSalidasPLC.LaserB;
SS.4 := gSalidasPLC.LaserC;
SS.11 := gSalidasPLC.LaserAA;		//A'
SS.12 := gSalidasPLC.LaserBB;		//B'
SS.13 := gSalidasPLC.LaserCC;		//C'

gSalidasPLC.SetaEmergenciaOUT1 := TRUE;
gSalidasPLC.SetaEmergenciaOUT2 := TRUE;

CAN_ENABLE(xEnable:=1,eChannel:=ifmdevice.CAN_CHANNEL.CHAN_0,eBaudrate:=250);

//---- Escribimos la variables estadoEframe con el estado en que estamos para enviar por CAN al AGV -----//
CASE gEstadoEframe OF
	Identificar:		
		estadoEframe := 0;
	Reposo:		
		IF (gEstadoCarga=cargado) THEN 
			estadoEframe := 1; 
		ELSE 
			estadoEframe := 2; 
		END_IF;
	Automatico:	
		estadoEframe := 3;
	Manual:		
		estadoEframe := 4;
	Degradado:	
		estadoEframe := 5;
	Reinicio:		
		estadoEframe := 6;
	Anomalia:		
		estadoEframe := 7;
END_CASE;

//-------------------------------------------------------------------------------------------//
//----------------------------Envio de informacion al AGV por CAN----------------------------//
//-------------------------------------------------------------------------------------------//
IF gEntradasPLC.SetaEmergenciaIN1 AND gEntradasPLC.SetaEmergenciaIN2 THEN
	gSalidasPLC.Seta_CAN := FALSE;
ELSE
	gSalidasPLC.Seta_CAN := TRUE;
END_IF

COMUNICACION_CAN.I_MatrizTX_AGV[0].0 := gSalidasPLC.Seta_CAN;
COMUNICACION_CAN.I_MatrizTX_AGV[0].1 := gEntradasPLC.ParadaPrecisaEFrame;
COMUNICACION_CAN.I_MatrizTX_AGV[0].2 := estadoEframe.0;
COMUNICACION_CAN.I_MatrizTX_AGV[0].3 := estadoEframe.1;
COMUNICACION_CAN.I_MatrizTX_AGV[0].4 := estadoEframe.2;
COMUNICACION_CAN.I_MatrizTX_AGV[0].5 := PosicionGrupo.0;
COMUNICACION_CAN.I_MatrizTX_AGV[0].6 := PosicionGrupo.1;
COMUNICACION_CAN.I_MatrizTX_AGV[0].7 := PosicionGrupo.2;

COMUNICACION_CAN.I_MatrizTX_AGV[1] := gSupS_MensajeAnom;

//-------------------------------------------------------------------------------------------//
//----------------------------------Comunicacion CAN Variador--------------------------------//
//-------------------------------------------------------------------------------------------//
IF SME_DRIVER THEN
	IF PrimerCiclo THEN
		C40.NumID:=1;
		C40.MatrizID[1]:=65;
		C41.RespuestasTotales[1]:=16#1F;        //----- Tiene que recibir informacion de 5 PDOs -----//
	END_IF;

	//----- Control potencia. Filtramos por estado para encendido secuenciado -----//
	TON_Reposo(IN:=(C41.ConsignaVariador[1]=0), PT:=T#1s);
	TON_InitializacionSME(IN:=TRUE, PT:=T#1.5s);
	C40.SafetyReleased := TRUE;
	C40.CORTE := C40.SafetyReleased AND TON_InitializacionSME.Q;

	//----- Parametrizacion -----//
	C41.LimitePar[1]:=INT_TO_WORD(SME_TORQUE);
	
	IF (AccionBrazo = M_Extender) OR (AccionBrazo = A_Extender) THEN
		C41.Atenuacion[1]:=100;
	ELSE
		C41.Atenuacion[1]:=100;
	END_IF
	
	//----- Rampa para llegar a la consigna deseada -----//
	TON_SalirLaser( IN:=AUX_SalirLaser, PT:=T#3S, ET => Tiempo_SalidaLaser);
	IF (NOT TON_SalirLaser.Q) AND (gEstadoEframe = Automatico)AND (LASER_AUX) THEN
		ConsignaVariador := gVelocidad;
	END_IF
	
	IF (NOT LASER_AUX) AND Reset_Consigna AND (gSalidasPlc.Consigna <> 0)  AND (gEstadoEframe = Automatico) THEN
		ConsignaVariador := 0;
		ConsignaA := 0;
		RampaTotal := 0;
		Reset_Consigna := FALSE;
	END_IF
	
	IF (NOT LASER_AUX) AND (ConsignaA <> gSalidasPlc.Consigna) THEN
		gRampaVelocidad := 1;
	ELSIF (NOT LASER_AUX) AND (gSalidasPlc.Consigna<10) AND (gSalidasPlc.Consigna>(-10)) THEN
		gRampaVelocidad := 2;
	ELSIF (NOT LASER_AUX) AND (ABS(gSalidasPlc.Consigna-ConsignaVariador)<20) THEN
		gRampaVelocidad := 3;
	ELSIF (NOT LASER_AUX) AND (NOT RampaCumplida) THEN
		gRampaVelocidad := 4;
	ELSIF LASER_AUX AND (gSalidasPlc.Consigna<10) AND (gSalidasPlc.Consigna>(-10)) THEN
		gRampaVelocidad := 5;
	END_IF
	
	CASE gRampaVelocidad OF
		1: // La velocidad de la consigna es distinta de la velocidad anterior
			RampaCumplida := FALSE;
			RampaTotal := (gSalidasPlc.Consigna-ConsignaA);
			AuxRampaLaser := FALSE;
			
		2: // Si la velocidad de la consigna es 0
			RampaCumplida := TRUE;
			ConsignaVariador := 0;
			AuxRampaLaser := FALSE;
			
		3: // Cuando la consigna deseada es atingida
			RampaCumplida := TRUE;
			ConsignaVariador := gSalidasPlc.Consigna;
			AuxRampaLaser := FALSE;
			
		4: // Cuando la rampa no es cumplida
			ConsignaVariador := ConsignaVariador + (RampaTotal/100);
			ConsignaVariadorA := ConsignaVariador;
			RampaA := RampaTotal;
			RestauroConsignaA := ConsignaA;
			AuxRampaLaser := FALSE;
			
		5: // Cuando se detecta láser y la consigan es 0
			IF (NOT AuxRampaLaser) THEN
				ConsignaVariadorA := ConsignaVariador;
				RampaA := RampaTotal;
				RestauroConsignaA := ConsignaA;
				AuxRampaLaser := TRUE;
			END_IF
			
			RampaCumplida := FALSE;
			ConsignaVariador := 0;
			ConsignaA := 0;
			RampaTotal := 0;
	END_CASE
	
	ConsignaA := gSalidasPlc.Consigna;

	//----- Comprova que esta todo bien y envia la velocidad -----//
	IF (C41.Estado[1]=6 AND C40.CORTE) THEN
		gRampaTotal := RampaTotal;
		gConsignaA := ConsignaA;
		gConsignaSalida := gSalidasPlc.Consigna;
		gEstadoRampa := RampaCumplida;
		gConsignaVariador := ConsignaVariador;
		C41.ConsignaVariador[1]:=ConsignaVariador;
	ELSE
		C41.ConsignaVariador[1]:=0;
	END_IF;

	//----- Magnetizacion y freno -----//
	IF C41.ConsignaVariador[1]<>0 THEN
		C41.MagnetizarMotor[1] := 1;
	ELSIF TON_Reposo.Q THEN
		C41.MagnetizarMotor[1] := 0;
	END_IF;

	C40(); //----- SME Llamada módulo principal -----//
END_IF;

//-------------------------------------------------------------------------------------------//
//-----------------------------------Comunicacion CAN Encoder--------------------------------//
//-------------------------------------------------------------------------------------------//
IF TON1.Q THEN
	IF AUX = 1 THEN
		MatrizEnvio1[0]:= 16#80;
		MatrizEnvio1[1]:= 0;
		MatrizEnvio1[2]:= 0;
		MatrizEnvio1[3]:= 0;
		MatrizEnvio1[4]:= 0;
		MatrizEnvio1[5]:= 0;
		MatrizEnvio1[6]:= 0;
		MatrizEnvio1[7]:= 0;
	
		CAN_TX1(xEnable:=TRUE, eChannel:=ifmdevice.CAN_CHANNEL.CHAN_2,usiDLC:=8, udiID:=16#0, aData:=MatrizEnvio1);
		
		AUX := 2;
	END_IF;
END_IF;

IF TON1.Q THEN
	IF AUX = 2 THEN
		MatrizEnvio2[0]:= 16#01;
		MatrizEnvio2[1]:= 0;
		MatrizEnvio2[2]:= 0;
		MatrizEnvio2[3]:= 0;
		MatrizEnvio2[4]:= 0;
		MatrizEnvio2[5]:= 0;
		MatrizEnvio2[6]:= 0;
		MatrizEnvio2[7]:= 0;
	
		CAN_TX1(xEnable:=TRUE, eChannel:=ifmdevice.CAN_CHANNEL.CHAN_2,usiDLC:=8, udiID:=16#0, aData:=MatrizEnvio2);
		
		AUX := 0;
	END_IF;
END_IF;

//----- Envio de informacion para el AGV -----//
COMUNICACION_CAN( I_OPERACION_CAN:=1 );

//----- Lectura de los valores del encoder de hilo -----//
Encoder_inicial := %ID135;
Encoder := %ID136;

END_PROGRAM

// StandardPLC/Application/CÓDIGO/Seguridades/Campos_Laser
PROGRAM Campos_Laser
VAR
END_VAR

(*//////////////////////////////////////////////////////////////////////////////////////////////////////////////////////////////////////////////////////////////////////////////////////////////////////////////////////////////////////////////////
Campos_Laser (PRG)                     

Description:	Definicion de los campos láser
				
///////////////////////////////////////////////////////////////////////////////////////////////////////////////////////////////////////////////////////////////////////////////////////////////////////////////////////////////////////////////////// *)

CASE Laser OF
	Bumper:
		gSalidasPLC.LaserA 	:= 0;
		gSalidasPLC.LaserB 	:= 0;
		gSalidasPLC.LaserC 	:= 0;
		gSalidasPLC.LaserAA := 1;
		gSalidasPLC.LaserBB := 1;
		gSalidasPLC.LaserCC := 1;
		
	Ext_sin_carga:
		gSalidasPLC.LaserA 	:= 0;
		gSalidasPLC.LaserB 	:= 1;
		gSalidasPLC.LaserC 	:= 0;
		gSalidasPLC.LaserAA := 1;
		gSalidasPLC.LaserBB := 0;
		gSalidasPLC.LaserCC := 1;
		
	Ext_con_carga_1600:
		gSalidasPLC.LaserA 	:= 0;
		gSalidasPLC.LaserB 	:= 0;
		gSalidasPLC.LaserC 	:= 1;
		gSalidasPLC.LaserAA := 1;
		gSalidasPLC.LaserBB := 1;
		gSalidasPLC.LaserCC := 0;
		
	Ext_con_carga_1800:
		gSalidasPLC.LaserA 	:= 0;
		gSalidasPLC.LaserB 	:= 1;
		gSalidasPLC.LaserC 	:= 1;
		gSalidasPLC.LaserAA := 1;
		gSalidasPLC.LaserBB := 0;
		gSalidasPLC.LaserCC := 0;
END_CASE

END_PROGRAM

// StandardPLC/Application/CÓDIGO/COMUNICACION_CAN
PROGRAM COMUNICACION_CAN
VAR_INPUT
	I_OPERACION_CAN			:BOOL;						//----- Seleccionar operación lectura/escritura del bus CAN -----//
	I_MatrizTX_AGV			:ARRAY [0..7] OF USINT;
END_VAR
VAR_OUTPUT
	O_MatrizRX_AGV			:ARRAY [0..7] OF USINT;
	O_EstadoCAN				:BYTE;
END_VAR
VAR
	CAN1_ComAGV				:COM00_DispositivoCAN_FB;
	
	PDO_ComAGV_TX			:DWORD;
	PDO_ComAGV_RX			:DWORD;
	
	i						:INT;
END_VAR

(*//////////////////////////////////////////////////////////////////////////////////////////////////////////////////////////////////////////////////////////////////////////////////////////////////////////////////////////////////////////////////
COMUNICACION_CAN (PRG)                     

Description:  	Módulo de la interface CAN con el AGV.
				Tenemos dos modos de operación:
					I_OPERACION_CAN := 0  -> leer datos CAN
					I_OPERACION_CAN := 1  -> escribir datos CAN
				                            				 
///////////////////////////////////////////////////////////////////////////////////////////////////////////////////////////////////////////////////////////////////////////////////////////////////////////////////////////////////////////////////// *)

IF PrimerCiclo THEN			// Configuraciones para la comunicacion
	//----- Asignacion PDOs -----//
	PDO_ComAGV_TX		:= 16#32;							//----- PDO 0x32 -----/
	PDO_ComAGV_RX		:= 16#28 + (PosicionGrupo/4);		//----- PDO	0x28 o 0x29 -----//
	
	//----- Configuracion Interfaces -----//	
	CAN1_ComAGV( 	I_ENABLE := FALSE,
					I_INTERFAZ_CAN := ifmDevice.CAN_CHANNEL.CHAN_0,
				    I_BAUDRATE := ifmDevice.CAN_BAUDRATE.KBAUD_250,
					I_ID_ENVIO := PDO_ComAGV_TX,
					I_ID_RECEPCION := PDO_ComAGV_RX );
ELSE	// OPERACION
	IF NOT I_OPERACION_CAN THEN
		//----- RECEPCION DE INFORMACION -----//
		CAN1_ComAGV( I_ENABLE:=TRUE, I_OPERACION:=1 );

		IF CAN1_ComAGV.O_ESTADO=16#F THEN		//----- Si no hay error actualizamos -----//
			O_MatrizRX_AGV := CAN1_ComAGV.O_MatrizRecepcion;
		ELSE
			FOR i:=0 TO 7 DO O_MatrizRX_AGV[i] := 0; END_FOR;
		END_IF;

	ELSE
		//----- ENVIO DE INFORMACION -----//
		CAN1_ComAGV( I_ENABLE:=TRUE, I_OPERACION:=2, I_MatrizEnvio:=I_MatrizTX_AGV );
	END_IF;

	//----- Mapeo anomalías -----//
	O_EstadoCAN.0 := CAN1_ComAGV.O_ESTADO.0;
	O_EstadoCAN.1 := CAN1_ComAGV.O_ESTADO.1;
END_IF;

END_PROGRAM

// StandardPLC/Application/CÓDIGO/Sub Comunicacion/COM00_DispositivoCAN_FB
FUNCTION_BLOCK COM00_DispositivoCAN_FB
VAR_INPUT
	I_ENABLE				:BOOL;
	I_OPERACION				:BYTE;
	I_INTERFAZ_CAN			:ifmDevice.CAN_CHANNEL;
	I_BAUDRATE				:ifmDevice.CAN_BAUDRATE;
	I_ID_ENVIO				:DWORD;
	I_ID_RECEPCION			:DWORD;

	I_MatrizEnvio			:ARRAY[0..7] OF USINT;
END_VAR

VAR_OUTPUT
	O_ESTADO				:BYTE;
	O_MatrizRecepcion		:ARRAY[0..7] OF USINT;
END_VAR

VAR
	//----- Variables interfaz CAN -----//	
	Interfaz_CAN			:ifmDevice.CAN_CHANNEL;
	Baudrate_CAN			:ifmDevice.CAN_BAUDRATE;
	IDEnvio					:DWORD;
	IDRecepcion				:DWORD;
	TON_HabilitarCom		:TON;
	CANX_ENABLE				:ifmRCAN.CAN_Enable;
	CANX_STATUS				:ifmRCAN.CAN_Status;
	CANX_RX					:ifmRCAN.CAN_Rx;
	CANX_TX					:ifmRCAN.CAN_Tx;

	//----- Variables para anomalías -----//	
	TON_CommRX				:TON;		//----- Tiempo sin comunicacion controlador -----//	
	CommRX					:BOOL;

	//----- Variables auxiliares -----//	
	MatrizVacia				:BOOL;
	aux_i					:INT;
	i						:INT;
END_VAR

(*//////////////////////////////////////////////////////////////////////////////////////////////////////////////////////////////////////////////////////////////////////////////////////////////////////////////////////////////////////////////////
COM00_DispositivoCAN_FB (FB)                     

Description:  	Módulo que implementa la interfaz CAN con variador Roboteq usando CAN2.

				Modos operacion:	        I_OPERACION := 1  --> leer datos CAN
						                            I_OPERACION := 2  --> escribir datos CAN	
	 
///////////////////////////////////////////////////////////////////////////////////////////////////////////////////////////////////////////////////////////////////////////////////////////////////////////////////////////////////////////////////// *)

//----- CONFIGURACION INTERNA -----//	
IF NOT I_ENABLE THEN
	Interfaz_CAN		:= I_INTERFAZ_CAN;
	Baudrate_CAN		:= I_BAUDRATE;
	IDRecepcion			:= I_ID_RECEPCION;
	IDEnvio				:= I_ID_ENVIO;
END_IF;

//----- Inicialización CAN -----//	
CANX_ENABLE( xEnable := I_ENABLE, eChannel := Interfaz_CAN, eBaudrate := Baudrate_CAN );

//----- Habilitar operaciones lectura/escritura, esperamos 2 segundos -----//	
TON_HabilitarCom( IN := I_ENABLE, PT := T#2s );

CANX_STATUS( xEnable := TON_HabilitarCom.Q, eChannel := Interfaz_CAN);

//----- Temporizador anomalía tiempo máximo sin comunicacion controlador -----//	
TON_CommRX( IN:=(CommRX AND TON_HabilitarCom.Q ), PT := T#500MS );
CommRX := I_ENABLE;

//----- Reset de las salidas -----//	
O_ESTADO := 16#F;

IF ( TON_HabilitarCom.Q ) THEN
	IF	CANX_STATUS.xError=FALSE THEN

		CASE I_OPERACION OF
			1: // RECEPCION
				CANX_RX( xEnable := TON_HabilitarCom.Q, eChannel := Interfaz_CAN, udiID := IDRecepcion );
				WHILE CANX_RX.uiAvailable>0 DO
					CommRX:=FALSE;
					O_MatrizRecepcion := CANX_RX.aData;
					CANX_RX( xEnable := TON_HabilitarCom.Q, eChannel := Interfaz_CAN, udiID := IDRecepcion );
				END_WHILE

			2: // ENVIO
				CANX_TX(xEnable := 1, eChannel := ifmDevice.CAN_CHANNEL.CHAN_0, udiID := IDEnvio, usiDLC := 8, aData := I_MatrizEnvio);
		END_CASE;
	END_IF;
END_IF;

//----- Anomalías dispositivo CAN -----//	
IF TON_CommRX.Q THEN		//----- Anomalía tiempo máximo sin comunicacion controlador superado -----//	
	O_ESTADO.0 := 0;
ELSE
	O_ESTADO.0 := 1;
END_IF;

IF ( TON_HabilitarCom.Q AND (CANX_STATUS.xError=TRUE) ) THEN	//----- Anomalía interfaz CAN -----//	
	O_ESTADO.1 := 0;
ELSE
	O_ESTADO.1 := 1;
END_IF;

END_FUNCTION_BLOCK

// StandardPLC/Application/CÓDIGO/Sub Comunicacion/C40
PROGRAM C40
VAR
	CAN_ENABLE1			:ifmRCAN.CAN_Enable;																		
	TONC40				:TON;
	TONC40b				:TON;
	ContarTONC40		:BOOL;
	Estado				:INT;
	EstadoA				:INT;
	I_ENABLE			:BOOL;
	aux_condicion		:BOOL;
	i					:INT;
END_VAR
VAR_INPUT
	Estado_Init			:INT;
	CORTE				:BOOL;
	NumID				:INT;
	MatrizID			:ARRAY[1..8] OF WORD;
	Reinicio			:BOOL;
	Rearme				:BOOL;
	SafetyReleased 		:BOOL;
END_VAR

(*/////////////////////////////////////////////////////////////////////////////////////////////////////////////////////////////////////////////////////////////////////////////////////////////////////////////////////////////////////////////////////
C40 (PRG)                   

Description:  Comunicacion con el variador por CAN - modulo general
			 
///////////////////////////////////////////////////////////////////////////////////////////////////////////////////////////////////////////////////////////////////////////////////////////////////////////////////////////////////////////////////// *)

TONC40(IN:=ContarTONC40, PT:=T#15S);
TONC40b(IN:=Estado=EstadoA, PT:=T#100ms);
EstadoA := Estado;
ContarTONC40 := 0;

//-------------------------------------------------------------------------------------------//
//------------------------------Reseteo estado cuando seta pulsada---------------------------//
//-------------------------------------------------------------------------------------------//
IF HabilitarVariador AND (NOT PrimerCiclo) THEN
	Estado := Estado_Init;	
END_IF

//-------------------------------------------------------------------------------------------//
//----------------------------------Inicializacion del variador------------------------------//
//-------------------------------------------------------------------------------------------//
CASE Estado OF
0:  // Espera respuesta  de los Variadores
	aux_condicion := 1;
	FOR i:=1 TO NumID DO
		IF C41.Estado[i] <> 1 THEN 
			aux_condicion := 0; 
		END_IF;
	END_FOR;

	IF CORTE THEN
		IF aux_condicion THEN
			Estado := 1;
		ELSIF TONC40.Q 	THEN
			Estado := -1;
		ELSIF NOT C41.TOF1_ON.Q THEN
			ContarTONC40 := 1;
		END_IF;
	END_IF;

1:  // Espera respuesta de estado correcto de los variadores
	aux_condicion := 1;
	FOR i:=1 TO NumID DO
		IF C41.Estado[i] <> 3 THEN 
			aux_condicion := 0; 
		END_IF;
	END_FOR;

	IF aux_condicion THEN
		Estado := 2;
	ELSIF TONC40.Q 	THEN
		Estado := -2;
	ELSE
		ContarTONC40 := 1;
	END_IF;

2:  // Orden de cargar condensadores, y espera a que la completen
	aux_condicion := 1;
	FOR i:=1 TO NumID DO
		IF C41.Estado[i] <> 5 THEN aux_condicion := 0; END_IF;
	END_FOR;

	IF aux_condicion THEN
		Estado := 3;
	ELSIF TONC40.Q 	THEN
		Estado := -3;
	ELSE
		ContarTONC40 := 1;
	END_IF;

3:  // Orden de activar el contactor que aplica la potencia, y espera a que la completen
	aux_condicion := 1;
	FOR i:=1 TO NumID DO
		IF C41.Estado[i] <> 6 THEN aux_condicion := 0; END_IF;
	END_FOR;

	IF aux_condicion THEN
		Estado := 4;
	ELSIF TONC40.Q 	THEN
		Estado := -4;
	ELSE
		ContarTONC40 := 1;
	END_IF;
4:  // Fin inicialización
	;
5:  // Reinicio Paso 1
	IF TONC40b.Q  AND CORTE THEN 
		Estado := 6; 
	END_IF;
6:  // Reinicio Paso 2
	IF TONC40b.Q THEN 
		Estado := 7; 
	END_IF;
7:  // Reinicio Paso 3
	IF TONC40b.Q THEN 
		Estado := 0; 
	END_IF;

ELSE  // Anomalía en la inicialización
	IF Rearme THEN 
		Estado := 5; 
	END_IF;
END_CASE;

CAN_ENABLE1(xEnable:=1,eChannel:=ifmdevice.CAN_CHANNEL.CHAN_1,eBaudrate:=250);

FOR i:=1 TO NumID DO
	C41.ID := MatrizID[i];
	C41.posi := i;
	C41();
END_FOR;

END_PROGRAM

// StandardPLC/Application/CÓDIGO/Sub Comunicacion/C41
PROGRAM C41
VAR
	CAN_RX_180					:ARRAY[1..8] OF ifmRCAN.CAN_Rx;																					
	CAN_RX_280					:ARRAY[1..8] OF ifmRCAN.CAN_Rx;	
	CAN_RX_380					:ARRAY[1..8] OF ifmRCAN.CAN_Rx;
	CAN_RX_480					:ARRAY[1..8] OF ifmRCAN.CAN_Rx;
	CAN_RX_6A0					:ARRAY[1..8] OF ifmRCAN.CAN_Rx;
	CAN_RX_680					:ARRAY[1..8] OF ifmRCAN.CAN_Rx;
	
	CAN_TX1						:ifmRCAN.CAN_Tx;	
	
	MatrizEnvio1A				:ARRAY[0..7] OF USINT;
	MatrizEnvio2A				:ARRAY[0..7] OF USINT;

	TOF1						:TOF;
	TONFirst					:TON;
	TOF1_ON						:TON;
	TONVariador					:TON;
	TONC41						:ARRAY[1..8] OF TON;
	ContarTONC41				:ARRAY[1..8] OF  BYTE;
	Estado						:ARRAY[1..8] OF BYTE;
	MatrizVacia					:ARRAY[1..8] OF BYTE;
	Valor						:ARRAY[1..8] OF INT;
	Fallo						:ARRAY[1..8] OF BYTE;
	TensionBusDC				:ARRAY[1..8] OF WORD;
	CorrienteBusDC				:ARRAY[1..8] OF WORD;
	TensionEntrada				:ARRAY[1..8] OF WORD;
	EntradaAnalogica1			:ARRAY[1..8] OF WORD;
	EntradaAnalogica2			:ARRAY[1..8] OF WORD;
	EntradaAnalogica3			:ARRAY[1..8] OF WORD;
	EntradaAnalogica4			:ARRAY[1..8] OF WORD;
	EntradaAnalogica5			:ARRAY[1..8] OF WORD;
	EntradaAnalogica6			:ARRAY[1..8] OF WORD;
	EntradaDigital				:ARRAY[1..8] OF DWORD := [0,16#F0F0F0F0,0,0,0,0,0,0];
	EstadoSalidas				:ARRAY[1..8] OF BYTE;
	Velocidad					:ARRAY[1..8] OF INT;
	Par							:ARRAY[1..8] OF WORD;
	TemperaturaMotor			:ARRAY[1..8] OF BYTE;
	TemperaturaVariador			:ARRAY[1..8] OF BYTE;
	EstadoMotor					:ARRAY[1..8] OF BYTE;
	CorrienteDriver1			:ARRAY[1..8] OF WORD;
	CorrienteDriver2			:ARRAY[1..8] OF WORD;
	CorrienteDriver3			:ARRAY[1..8] OF WORD;
	TONDriver1					:ARRAY[1..8] OF TON;
	TONDriver2					:ARRAY[1..8] OF TON;
	TONDriver3					:ARRAY[1..8] OF TON;
	TON1						:ARRAY[1..8] OF TON;
	TON2						:ARRAY[1..8] OF TON;
	TON3						:ARRAY[1..8] OF TON;
	Contar1						:ARRAY[1..8] OF BOOL;
	Contar2						:ARRAY[1..8] OF BOOL;
	Contar3						:ARRAY[1..8] OF BOOL;
	MatrizVaciaR				:ARRAY[1..8] OF USINT;
	
	EstadoRX_Variador 			:BYTE;
	Anomalia_Variador 			:BYTE;
END_VAR
VAR_INPUT
	ID							:WORD;
	posi						:INT;
	RespuestasTotales			:ARRAY[1..8] OF BYTE;
	ConsignaVariador			:ARRAY[1..8] OF REAL;
	ConsignaVariador2			:ARRAY[1..8] OF REAL;
	Driver1						:ARRAY[1..8] OF BOOL;
	Driver2						:ARRAY[1..8] OF BOOL;
	Driver3						:ARRAY[1..8] OF BOOL;
	Driver1fijo					:ARRAY[1..8] OF BOOL;
	Driver2fijo					:ARRAY[1..8] OF BOOL;
	Driver3fijo					:ARRAY[1..8] OF BOOL;
	Driver1porcentaje			:ARRAY[1..8] OF REAL;
	Driver2porcentaje			:ARRAY[1..8] OF REAL;
	Driver3porcentaje			:ARRAY[1..8] OF REAL;
	Driver1Vmax					:ARRAY[1..8] OF REAL;
	Driver2Vmax					:ARRAY[1..8] OF REAL;
	Driver3Vmax					:ARRAY[1..8] OF REAL;
	LimitePar					:ARRAY[1..8] OF WORD;
	Atenuacion					:ARRAY[1..8] OF BYTE;
	MagnetizarMotor				:ARRAY[1..8] OF BOOL;
	SalidasDigitales			:ARRAY[1..8] OF BYTE;
	MatrizEnvio AT %MW750		:ARRAY[0..7] OF BYTE;
	
	Aux_real 					:REAL;							
							
	MatrizRecepcion				:ARRAY[0..7] OF USINT;
END_VAR

(*/////////////////////////////////////////////////////////////////////////////////////////////////////////////////////////////////////////////////////////////////////////////////////////////////////////////////////////////////////////////////////
C41 (PRG)                   

Description:  Comunicacion con el variador por CAN
			 
///////////////////////////////////////////////////////////////////////////////////////////////////////////////////////////////////////////////////////////////////////////////////////////////////////////////////////////////////////////////////// *)

TONFirst(IN:=NOT PrimerCiclo, PT:=T#2S);
TOF1_ON(IN:=PrimerCiclo, PT:=T#2S);

//----- Para iniciar la recepcion esperar unos 2 sg, primero a 1 y despues de 2 segundos 0 -----//
CAN_RX_180[posi](xEnable:=1,eChannel:=ifmdevice.CAN_CHANNEL.CHAN_1,udiID:=16#180+ID);
CAN_RX_280[posi](xEnable:=1,eChannel:=ifmdevice.CAN_CHANNEL.CHAN_1,udiID:=16#280+ID);
CAN_RX_380[posi](xEnable:=1,eChannel:=ifmdevice.CAN_CHANNEL.CHAN_1,udiID:=16#380+ID);
CAN_RX_480[posi](xEnable:=1,eChannel:=ifmdevice.CAN_CHANNEL.CHAN_1,udiID:=16#480+ID);
CAN_RX_6A0[posi](xEnable:=1,eChannel:=ifmdevice.CAN_CHANNEL.CHAN_1,udiID:=16#6A0+ID);
CAN_RX_680[posi](xEnable:=1,eChannel:=ifmdevice.CAN_CHANNEL.CHAN_1,udiID:=16#680+ID);

MatrizEnvio := MatrizVacia;

CASE C40.Estado OF
0:		MatrizEnvio[1] := 0;
1: 		MatrizEnvio[0] := 2;
2:		MatrizEnvio[0] := 4;
3,4:	MatrizEnvio[0] := 6;
5:		MatrizEnvio[0] := 1;	MatrizEnvio[1] := 0;
6:		MatrizEnvio[0] := 1; 	MatrizEnvio[1] := 32;			//----- Requiere un primero reset de Sw -----//
7:		MatrizEnvio[0] := 1; 	MatrizEnvio[1] := 64;			//----- Requiere un segundo reset de Sw -----//
END_CASE;

MatrizEnvio[1] := SalidasDigitales[posi];

TON1[posi](IN:=Contar1[posi], PT:=T#80ms+INT_TO_TIME(posi*10));
Contar1[posi] := 1;
IF NOT TOF1_ON.Q THEN
	IF TON1[posi].Q OR MatrizEnvio[0]<>MatrizEnvio1A[0] OR MatrizEnvio[1]<>MatrizEnvio1A[1] OR MatrizEnvio[2]<>MatrizEnvio1A[2] OR MatrizEnvio[3]<>MatrizEnvio1A[3] OR MatrizEnvio[4]<>MatrizEnvio1A[4] OR MatrizEnvio[5]<>MatrizEnvio1A[5] OR MatrizEnvio[6]<>MatrizEnvio1A[6] OR MatrizEnvio[7]<>MatrizEnvio1A[7] THEN
		CAN_TX1(xEnable:=TRUE, eChannel:=ifmdevice.CAN_CHANNEL.CHAN_1,usiDLC:=8, udiID:=16#200+ID, aData:=MatrizEnvio1A);
		
		MatrizEnvio1A[0] := BYTE_TO_USINT(MatrizEnvio[0]);
		MatrizEnvio1A[1] := BYTE_TO_USINT(MatrizEnvio[1]);
		MatrizEnvio1A[2] := BYTE_TO_USINT(MatrizEnvio[2]);
		MatrizEnvio1A[3] := BYTE_TO_USINT(MatrizEnvio[3]);				//----- Solo la MatrizEnvio1A[0] y la MatrizEnvio1A[1] van hacer transmission de dados -----//
		MatrizEnvio1A[4] := BYTE_TO_USINT(MatrizEnvio[4]);
		MatrizEnvio1A[5] := BYTE_TO_USINT(MatrizEnvio[5]);
		MatrizEnvio1A[6] := BYTE_TO_USINT(MatrizEnvio[6]);
		MatrizEnvio1A[7] := BYTE_TO_USINT(MatrizEnvio[7]);
		
		Contar1[posi] := 0;
	END_IF;
END_IF;

MatrizEnvio := MatrizVacia;

MatrizEnvio[0] := UINT_TO_BYTE(INT_TO_UINT(REAL_TO_INT(ConsignaVariador[posi])) MOD 16#100);
MatrizEnvio[1] := UINT_TO_BYTE(INT_TO_UINT(REAL_TO_INT(ConsignaVariador[posi])) /16#100);
MatrizEnvio[2] := WORD_TO_BYTE(LimitePar[posi] MOD 16#100);
MatrizEnvio[3] := WORD_TO_BYTE(LimitePar[posi] /16#100);
MatrizEnvio[4] := Atenuacion[posi];
MatrizEnvio[5].0 := 1;													//----- Modo control velocidad -----/
MatrizEnvio[5].2 := MagnetizarMotor[posi];
MatrizEnvio[5].3 := 1;

TON2[posi](IN:=Contar2[posi], PT:=T#90ms+INT_TO_TIME(posi*10));
Contar2[posi] := 1;
IF NOT TOF1_ON.Q THEN
	IF TON2[posi].Q OR MatrizEnvio[0]<>MatrizEnvio2A[0] OR MatrizEnvio[1]<>MatrizEnvio2A[1] OR MatrizEnvio[2]<>MatrizEnvio2A[2] OR MatrizEnvio[3]<>MatrizEnvio2A[3] OR MatrizEnvio[4]<>MatrizEnvio2A[4] OR MatrizEnvio[5]<>MatrizEnvio2A[5] OR MatrizEnvio[6]<>MatrizEnvio2A[6] OR MatrizEnvio[7]<>MatrizEnvio2A[7] THEN
		CAN_TX1(xEnable:=1, eChannel:=ifmdevice.CAN_CHANNEL.CHAN_1,usiDLC:=8, udiID:=16#300+ID, aData:=MatrizEnvio2A);
		
		MatrizEnvio2A[0] := MatrizEnvio[0];
		MatrizEnvio2A[1] := MatrizEnvio[1];
		MatrizEnvio2A[2] := MatrizEnvio[2];
		MatrizEnvio2A[3] := MatrizEnvio[3];					//----- Solo la MatrizEnvio2A[6] y la MatrizEnvio2A[7] no van hacer transmission de dados -----//
		MatrizEnvio2A[4] := MatrizEnvio[4];
		MatrizEnvio2A[5] := MatrizEnvio[5];
		MatrizEnvio2A[6] := MatrizEnvio[6];
		MatrizEnvio2A[7] := MatrizEnvio[7];
		
		Contar2[posi] := 0;
	END_IF;
END_IF;

MatrizEnvio := MatrizVacia;

MatrizRecepcion := MatrizVaciaR;

WHILE CAN_Rx_180[posi].uiAvailable > 0 DO	

	MatrizRecepcion:=CAN_Rx_180[posi].aData;

	IF CAN_Rx_180[posi].uiAvailable=1 THEN	
		Estado[posi]:= MatrizRecepcion[0];
		Fallo[posi]:= MatrizRecepcion[1];
		TensionBusDC[posi] := BYTE_TO_WORD(MatrizRecepcion[2])+BYTE_TO_WORD(MatrizRecepcion[3])*16#100;
		CorrienteBusDC[posi]:= BYTE_TO_WORD(MatrizRecepcion[4])+BYTE_TO_WORD(MatrizRecepcion[5])*16#100;
		TensionEntrada[posi]:=BYTE_TO_WORD(MatrizRecepcion[6])+BYTE_TO_WORD(MatrizRecepcion[7])*16#100;

		ContarTONC41[posi].0 := 1;
	END_IF;

	CAN_RX_180[posi](xEnable:=1,eChannel:=ifmdevice.CAN_CHANNEL.CHAN_1,udiID:=16#180+ID);
	
END_WHILE;

MatrizRecepcion := MatrizVaciaR;

WHILE CAN_Rx_280[posi].uiAvailable>0 DO	

	MatrizRecepcion:=CAN_Rx_280[posi].aData;

	IF CAN_Rx_280[posi].uiAvailable=1 THEN	
		EntradaAnalogica1[posi] := BYTE_TO_WORD(MatrizRecepcion[0])+BYTE_TO_WORD(MatrizRecepcion[1])*16#100;
		EntradaAnalogica2[posi] :=BYTE_TO_WORD(MatrizRecepcion[2])+BYTE_TO_WORD(MatrizRecepcion[3])*16#100;
		EntradaAnalogica3[posi] := BYTE_TO_WORD(MatrizRecepcion[4])+BYTE_TO_WORD(MatrizRecepcion[5])*16#100;
		EntradaAnalogica4[posi] := BYTE_TO_WORD(MatrizRecepcion[6])+BYTE_TO_WORD(MatrizRecepcion[7])*16#100;

		ContarTONC41[posi].1 := 1;
	END_IF;
	
	CAN_RX_280[posi](xEnable:=1,eChannel:=ifmdevice.CAN_CHANNEL.CHAN_1,udiID:=16#280+ID);
	
END_WHILE;

MatrizRecepcion := MatrizVaciaR;

WHILE CAN_Rx_380[posi].uiAvailable>0 DO

	MatrizRecepcion:=CAN_Rx_380[posi].aData;

	IF CAN_Rx_380[posi].uiAvailable=1 THEN	
		EntradaAnalogica5[posi] := BYTE_TO_WORD(MatrizRecepcion[0])+BYTE_TO_WORD(MatrizRecepcion[1])*16#100;
		EntradaAnalogica6[posi] := BYTE_TO_WORD(MatrizRecepcion[2])+BYTE_TO_WORD(MatrizRecepcion[3])*16#100;
		EntradaDigital[posi]:= BYTE_TO_DWORD(MatrizRecepcion[4])+BYTE_TO_DWORD(MatrizRecepcion[5])*16#100;
		EntradaDigital[posi]:= EntradaDigital[posi]+BYTE_TO_DWORD(MatrizRecepcion[6])*16#10000;
		EstadoSalidas[posi] := MatrizRecepcion[7];

		ContarTONC41[posi].2 := 1;
	END_IF;
	
	CAN_RX_380[posi](xEnable:=1,eChannel:=ifmdevice.CAN_CHANNEL.CHAN_1,udiID:=16#380+ID);
END_WHILE;

MatrizRecepcion := MatrizVaciaR;
																			
WHILE CAN_Rx_480[posi].uiAvailable>0 DO																			

	MatrizRecepcion:=CAN_Rx_480[posi].aData;					
																			
	IF CAN_Rx_480[posi].uiAvailable=1 THEN			
		IF MatrizRecepcion[1]>16#7F THEN
			Velocidad[posi]:=DINT_TO_INT(BYTE_TO_DINT(MatrizRecepcion[0])+BYTE_TO_DINT(MatrizRecepcion[1])*16#100-16#10000);
		ELSE
			Velocidad[posi]:=BYTE_TO_INT(MatrizRecepcion[0])+BYTE_TO_INT(MatrizRecepcion[1])*16#100;
		END_IF;
		Par[posi]:= BYTE_TO_WORD(MatrizRecepcion[2])+BYTE_TO_WORD(MatrizRecepcion[3])*16#100;
		TemperaturaMotor[posi]:=MatrizRecepcion[4] - 40;
		TemperaturaVariador[posi]:=MatrizRecepcion[5] - 40;
		EstadoMotor[posi]:=MatrizRecepcion[7];

		ContarTONC41[posi].3 := 1;
	END_IF;
											
	CAN_RX_480[posi](xEnable:=1,eChannel:=ifmdevice.CAN_CHANNEL.CHAN_1,udiID:=16#480+ID);
END_WHILE;

MatrizRecepcion := MatrizVaciaR;
											
WHILE CAN_Rx_6A0[posi].uiAvailable>0 DO	

	MatrizRecepcion:=CAN_Rx_6A0[posi].aData;

	IF CAN_Rx_6A0[posi].uiAvailable=1 THEN										
		CorrienteDriver1[posi]:=BYTE_TO_WORD(MatrizRecepcion[0])+BYTE_TO_WORD(MatrizRecepcion[1])*16#100;
		CorrienteDriver2[posi]:=BYTE_TO_WORD(MatrizRecepcion[2])+BYTE_TO_WORD(MatrizRecepcion[3])*16#100;
		CorrienteDriver3[posi]:=BYTE_TO_WORD(MatrizRecepcion[4])+BYTE_TO_WORD(MatrizRecepcion[5])*16#100;

		ContarTONC41[posi].4 := 1;
	END_IF;
																	
	CAN_RX_6A0[posi](xEnable:=1,eChannel:=ifmdevice.CAN_CHANNEL.CHAN_1,udiID:=16#6A0+ID);	
END_WHILE;

MatrizRecepcion := MatrizVaciaR;
																				
WHILE CAN_Rx_680[posi].uiAvailable>0 DO	

	MatrizRecepcion:=CAN_Rx_680[posi].aData;

	ContarTONC41[posi].5 := 1;
	
	CAN_RX_680[posi](xEnable:=1,eChannel:=ifmdevice.CAN_CHANNEL.CHAN_1,udiID:=16#680+ID);
END_WHILE;

//----- tiempo espera respuesta inverter -----//	
TONC41[posi](IN:=ContarTONC41[posi]<>RespuestasTotales[posi] AND NOT TOF1_ON.Q, PT:=T#300MS);
IF TONC41[posi].Q THEN
	Valor[posi]:=-1;	 //----- no ha respondido el variador -----//	
ELSE
	Valor[posi]:=0;
END_IF;

IF (Estado[posi]>3) AND (Estado[posi] <> 7) AND (NOT SetaPulsada_AUX) THEN
	gSalidasPLC.Contactor := TRUE;
	gSalidasPLC.Contactor2 := TRUE;
ELSE 
	gSalidasPLC.Contactor := FALSE;
	gSalidasPLC.Contactor2 := FALSE;
END_IF;

IF ContarTONC41[posi]=RespuestasTotales[posi] THEN 
	ContarTONC41[posi]:=0;	
END_IF;

TONVariador(IN:= (Estado[posi]>6 OR C40.Estado <0), PT:=T#20S);

IF TONVariador.Q AND (NOT RESET) THEN					//----- Anomalía sin respuesta del variador -----//	
	EstadoRX_Variador.0 := 0;
ELSE
	EstadoRX_Variador.0 := 1;
END_IF;

IF Estado[posi] = 7 THEN                //----- Indica si el variador esta en estado de anomalia -----//	
	Anomalia_Variador.0 := 0;
ELSE
	Anomalia_Variador.0 := 1;
END_IF

END_PROGRAM

// StandardPLC/Application/CÓDIGO/PARAMETRIZACION
PROGRAM PARAMETRIZACION
VAR
	
END_VAR

(*/////////////////////////////////////////////////////////////////////////////////////////////////////////////////////////////////////////////////////////////////////////////////////////////////////////////////////////////////////////////////
PARAMETRIZACION (PRG)                     

Description:  Parametrizacion de variables globales
///////////////////////////////////////////////////////////////////////////////////////////////////////////////////////////////////////////////////////////////////////////////////////////////////////////////////////////////////////////////////// *)

//-------------------------------------------------------------------------------------------//
//--------------------------Parametros de configuracion del variador-------------------------//
//-------------------------------------------------------------------------------------------//
SME_DRIVER := 1;
SME_TORQUE := 32000;					//----- Par máximo 32000 -----//
SME_SPEEDRPM_INIT := 0;					//----- Velocidad telescópico rpm cuando está retraido -----//
SME_SPEEDRPM_MANUAL:= 600;				//----- Velocidad telescópico en modo manual -----//

//-------------------------------------------------------------------------------------------//
//                             Tramos de las velocidades:                                    //
// 3 TRAMOS:                                                                                 //
//             TRAMO1                    TRAMO2                   TRAMO3                     //
//    |------------------------|------------------------|------------------------|           //
//  Inicio                                                                    Extendido      //
//                                                                                           //
// 2 TRAMOS:                                                                                 //
//                    TRAMO1                                TRAMO2                           //
//    |-------------------------------------|------------------------------------|           //
//  Inicio                                                                    Extendido      //
//-------------------------------------------------------------------------------------------//

//----- Velocidades de los distintos tramos para extension cargado -----//
SME_SPEEDRPM_E_Cargado_Tramo1 := 800;          //550
SME_SPEEDRPM_E_Cargado_Tramo2 := 1000;         //800
SME_SPEEDRPM_E_Cargado_Tramo3 := 600;          //350

//----- Velocidades de los distintos tramos para extension descargado -----//
SME_SPEEDRPM_E_Descargado_Tramo1 := 1500;
SME_SPEEDRPM_E_Descargado_Tramo2 := 1200;
SME_SPEEDRPM_E_Descargado_Tramo3 := 500;


//----- Velocidades de los distintos tramos para recoja descargado -----//
SME_SPEEDRPM_R_Descargado_Tramo1 :=600;          //800
SME_SPEEDRPM_R_Descargado_Tramo2 := 1500;        //1000

//----- Velocidades de los distintos tramos para recoja cargado -----//
SME_SPEEDRPM_R_Cargado_Tramo1 := 600;          
SME_SPEEDRPM_R_Cargado_Tramo2 := 1200;          
SME_SPEEDRPM_R_Cargado_Tramo3 := 800;          


//-------------------------------------------------------------------------------------------//
//------------------------Valores de configuracion del Encoder de Hilo-----------------------//
//-------------------------------------------------------------------------------------------//
Recorrido_Standard := 49000; 					//----- Variable que indica el recogido del brazo del E-Frame -----//

E_Tramo1 := gEncoder_Absoluto - 16000;			//----- Calculo del valor del encoder para el tramo1 teniendo en cuenta el valor absoluto del E-Frame -----//
E_Tramo2 := gEncoder_Absoluto - 35000;			//----- Calculo del valor del encoder para el tramo2 teniendo en cuenta el valor absoluto del E-Frame -----//

